{attribute 'qualified_only'}
VAR_GLOBAL  (* GVL_IO *)
  DI_Security_Open : ARRAY[1..GVL_CONSTANTS.C_MAX_SECURITY_SENSORS] OF BOOL;
  DI_Security_Glass : ARRAY[1..GVL_CONSTANTS.C_MAX_SECURITY_SENSORS] OF BOOL;
  DI_Security_2F_Group : BOOL;
  DI_Flood_Sensors : ARRAY[1..GVL_CONSTANTS.C_MAX_FLOOD_SENSORS] OF BOOL;
  DI_Manifold_End_Switches : ARRAY[1..GVL_CONSTANTS.C_MAX_MANIFOLDS] OF BOOL;
  AO_Manifold_Valves : ARRAY[1..GVL_CONSTANTS.C_MAX_MANIFOLDS] OF UINT;
  DO_Manifold_Pumps : ARRAY[1..GVL_CONSTANTS.C_MAX_MANIFOLDS] OF BOOL;
  AI_Manifold_Currents : ARRAY[1..GVL_CONSTANTS.C_MAX_MANIFOLDS] OF INT;
  AI_Manifold_Pressures : ARRAY[1..GVL_CONSTANTS.C_MAX_MANIFOLDS] OF INT;
  AI_Manifold_Temps_Supply : ARRAY[1..GVL_CONSTANTS.C_MAX_MANIFOLDS] OF ST_Owen_Analog_Value;
  AI_Manifold_Temps_Return : ARRAY[1..GVL_CONSTANTS.C_MAX_MANIFOLDS] OF INT;
  AO_Supply_Fans : ARRAY[1..GVL_CONSTANTS.C_MAX_SUPPLY_FANS] OF UINT;
  AO_Exhaust_Fans : ARRAY[1..GVL_CONSTANTS.C_MAX_EXHAUST_FANS] OF UINT;
  AO_Lighting_Levels : ARRAY[1..GVL_CONSTANTS.C_MAX_LIGHT_ZONES] OF UINT;
  AO_Blinds_Positions : ARRAY[1..GVL_CONSTANTS.C_MAX_BLINDS] OF UINT;
  AI_Supply_Temps : ARRAY[1..GVL_CONSTANTS.C_MAX_SUPPLY_TEMPS] OF ST_Owen_Analog_Value;
  AI_Boiler_Modulation : ARRAY[1..GVL_CONSTANTS.C_MAX_BOILERS] OF INT;
  AI_Boiler_Flame_Status : ARRAY[1..GVL_CONSTANTS.C_MAX_BOILERS] OF BOOL;
  DI_Boiler_Error : ARRAY[1..GVL_CONSTANTS.C_MAX_BOILERS] OF BOOL;
  AI_Methane_LEL : ARRAY[1..GVL_CONSTANTS.C_MAX_METHANE_SENSORS] OF ST_Owen_Analog_Value;
  AI_CO_PPM : ARRAY[1..GVL_CONSTANTS.C_MAX_CO_SENSORS] OF REAL;
  DI_Smoke_Sensors : ARRAY[1..GVL_CONSTANTS.C_MAX_SMOKE_SENSORS] OF BOOL;
  AI_Temp_Outdoor : ST_Owen_Analog_Value;
  AI_Floor_Temps : ARRAY[1..GVL_CONSTANTS.C_MAX_ZONES] OF REAL;
  AI_Room_Temps : ARRAY[1..GVL_CONSTANTS.C_MAX_ZONES] OF REAL;
  AI_Room_Hum : ARRAY[1..GVL_CONSTANTS.C_MAX_ZONES] OF REAL;
  AI_Room_CO2 : ARRAY[1..GVL_CONSTANTS.C_MAX_ZONES] OF REAL;
  DO_Zone_Valves : ARRAY[1..GVL_CONSTANTS.C_MAX_HEATING_CIRCUITS] OF BOOL;
  AI_DHW_Temp : REAL;
  AI_DHW_Pressure : REAL;
  DO_DHW_Heating_Pump : BOOL;
  DO_DHW_Circ_Pump : BOOL;
  DO_Backup_Circulation_Pump : BOOL;
  DO_Electric_Heater_Enable : BOOL;
  DI_Lighting_Switches : ARRAY[1..GVL_CONSTANTS.C_MAX_LIGHT_ZONES] OF BOOL;
  DI_Socket_Switches : ARRAY[1..GVL_CONSTANTS.C_MAX_SOCKETS] OF BOOL;
  DI_Motion_Sensors : ARRAY[1..GVL_CONSTANTS.C_MAX_LIGHT_ZONES] OF BOOL;
  DO_Sockets : ARRAY[1..GVL_CONSTANTS.C_MAX_SOCKETS] OF BOOL;
  DO_Gas_Valve_Close : BOOL;
  DO_Water_Valve_35_Close : BOOL;
  DO_Water_Valve_36_Close : BOOL;
  AI_Water_Valve_35_Current : REAL;
  AI_Water_Valve_36_Current : REAL;
  DI_Power_OK : BOOL;
  DO_Gas_Siren : BOOL;
  DO_Fire_Siren : BOOL;
  DO_Security_Siren : BOOL;
  DO_Pump_Main_Enable : BOOL;
  DO_Gate_Open : BOOL;
  DO_Wicket_Open : BOOL;
  DO_Lock_1_Open : BOOL;
  DO_Lock_1_Close : BOOL;
  DO_Lock_2_Open : BOOL;
  DO_Lock_2_Close : BOOL;
  DI_Partner_Pulse : BOOL;
  DI_Partner_Active : BOOL;
  DO_Heartbeat_Pulse : BOOL;
  DO_Active_Status : BOOL;
  DI_Module_1_Heartbeat : BOOL;
  DI_Module_2_Heartbeat : BOOL;
  DI_Backup_Circulation_Pump_Feedback : BOOL;
  DI_Electric_Heater_Feedback : BOOL;
  DI_Water_Zone_Open_FB : ARRAY[1..GVL_CONSTANTS.C_MAX_WATER_ZONES] OF BOOL;
  DI_Water_Zone_Close_FB : ARRAY[1..GVL_CONSTANTS.C_MAX_WATER_ZONES] OF BOOL;
  DO_Water_Zone_Enable : ARRAY[1..GVL_CONSTANTS.C_MAX_WATER_ZONES] OF BOOL;
END_VAR

VAR_GLOBAL  (* GVL_Safety_Selector *)
  G_Use_Shadow_CO : BOOL := FALSE;
  G_Use_Shadow_Methane : BOOL := FALSE;
  G_Use_Shadow_Smoke : BOOL := FALSE;
  G_CO_Effective : REAL;
  G_Methane_Effective : REAL;
  G_Smoke_Effective : BOOL;
  G_CO_Shadow_Max_Diff : REAL := 5.0;
  G_Methane_Shadow_Max_Diff : REAL := 5.0;
  G_Block_Shadow_On_Mismatch : BOOL := TRUE;
  G_Shadow_Unstable_Cycles_Limit : INT := 5;
  G_CO_Shadow_Recovery_Diff : REAL := 2.0;
  G_Methane_Shadow_Recovery_Diff : REAL := 2.0;
  G_CO_Stable_Counter : INT := 0;
  G_Methane_Stable_Counter : INT := 0;
  G_Smoke_Stable_Counter : INT := 0;
  G_CO_Unstable_Counter : INT := 0;
  G_Methane_Unstable_Counter : INT := 0;
  G_Smoke_Unstable_Counter : INT := 0;
  G_CO_Effective_Array : ARRAY[1..GVL_CONSTANTS.C_MAX_CO_SENSORS] OF REAL;
  G_Methane_Effective_Array : ARRAY[1..GVL_CONSTANTS.C_MAX_METHANE_SENSORS] OF REAL;
  G_Smoke_Effective_Array : ARRAY[1..GVL_CONSTANTS.C_MAX_SMOKE_SENSORS] OF BOOL;
END_VAR

{attribute 'qualified_only'}
VAR_GLOBAL  (* GVL_STATE *)
  G_Floor_Temps : ARRAY[1..GVL_CONSTANTS.C_MAX_HEATING_CIRCUITS] OF REAL;
  G_Room_Temps : ARRAY[1..GVL_CONSTANTS.C_MAX_ZONES] OF REAL;
  G_Last_Valid_Room_Temps : ARRAY[1..GVL_CONSTANTS.C_MAX_ZONES] OF REAL;
  G_Last_Valid_Floor_Temps : ARRAY[1..GVL_CONSTANTS.C_MAX_HEATING_CIRCUITS] OF REAL;
  G_Temp_Sensor_Fault : ARRAY[1..GVL_CONSTANTS.C_MAX_ZONES] OF BOOL;
  G_Floor_Temp_Sensor_Fault : ARRAY[1..GVL_CONSTANTS.C_MAX_HEATING_CIRCUITS] OF BOOL;
  G_Room_Hum : ARRAY[1..GVL_CONSTANTS.C_MAX_ZONES] OF REAL;
  G_Room_CO2 : ARRAY[1..GVL_CONSTANTS.C_MAX_ZONES] OF REAL;
  G_Motion_Sensors : ARRAY[1..GVL_CONSTANTS.C_MAX_LIGHT_ZONES] OF BOOL;
  G_Door_Sensors : ARRAY[1..GVL_CONSTANTS.C_MAX_DOOR_SENSORS] OF BOOL;
  G_Window_Sensors : ARRAY[1..GVL_CONSTANTS.C_MAX_ZONES] OF BOOL;
  G_Water_Sensors : ARRAY[1..GVL_CONSTANTS.C_MAX_FLOOD_SENSORS] OF BOOL;
  G_Flood_Warning : ARRAY[1..GVL_CONSTANTS.C_MAX_FLOOD_SENSORS] OF BOOL;
  G_Flood_Alarm : ARRAY[1..GVL_CONSTANTS.C_MAX_FLOOD_SENSORS] OF BOOL;
  G_Flood_Warning_Rise : ARRAY[1..GVL_CONSTANTS.C_MAX_FLOOD_SENSORS] OF BOOL;
  G_Flood_Alarm_Rise : ARRAY[1..GVL_CONSTANTS.C_MAX_FLOOD_SENSORS] OF BOOL;
  G_Flood_Alarm_Fall : ARRAY[1..GVL_CONSTANTS.C_MAX_FLOOD_SENSORS] OF BOOL;
  G_Smoke_Sensors : ARRAY[1..GVL_CONSTANTS.C_MAX_SMOKE_SENSORS] OF BOOL;
  G_Methane_Sensors : ARRAY[1..GVL_CONSTANTS.C_MAX_METHANE_SENSORS] OF REAL;
  G_CO_Sensors : ARRAY[1..GVL_CONSTANTS.C_MAX_CO_SENSORS] OF REAL;
  G_Manifold_Pressures : ARRAY[1..GVL_CONSTANTS.C_MAX_MANIFOLDS] OF REAL;
  G_Manifold_Currents : ARRAY[1..GVL_CONSTANTS.C_MAX_MANIFOLDS] OF REAL;
  G_Predictive_Pump_Pressure_Drop : ARRAY[1..GVL_CONSTANTS.C_MAX_MANIFOLDS] OF BOOL;
  G_Predictive_Pump_Current_Rise : ARRAY[1..GVL_CONSTANTS.C_MAX_MANIFOLDS] OF BOOL;
  G_Manifold_T_Supply : ARRAY[1..GVL_CONSTANTS.C_MAX_MANIFOLDS] OF REAL;
  G_Manifold_T_Return : ARRAY[1..GVL_CONSTANTS.C_MAX_MANIFOLDS] OF REAL;
  G_Boiler_Flame : ARRAY[1..GVL_CONSTANTS.C_MAX_BOILERS] OF BOOL;
  G_Boiler_Error : ARRAY[1..GVL_CONSTANTS.C_MAX_BOILERS] OF BOOL;
  G_Boiler_OT_Online : ARRAY[1..GVL_CONSTANTS.C_MAX_BOILERS] OF BOOL;
  G_Boiler_OT_Command_Ack : ARRAY[1..GVL_CONSTANTS.C_MAX_BOILERS] OF BOOL;
  G_Boiler_OT_Command_Timeout : ARRAY[1..GVL_CONSTANTS.C_MAX_BOILERS] OF BOOL;
  G_Boiler_OT_Heartbeat_Timeout : ARRAY[1..GVL_CONSTANTS.C_MAX_BOILERS] OF BOOL;
  G_Boiler_OT_Adapter_Error : ARRAY[1..GVL_CONSTANTS.C_MAX_BOILERS] OF BOOL;
  G_Boiler_OT_Heartbeat_Age_MS : ARRAY[1..GVL_CONSTANTS.C_MAX_BOILERS] OF UDINT;
  G_Boiler_OT_Command_Age_MS : ARRAY[1..GVL_CONSTANTS.C_MAX_BOILERS] OF UDINT;
  G_Boiler_OT_Adapter_State : ARRAY[1..GVL_CONSTANTS.C_MAX_BOILERS] OF E_OpenTherm_Adapter_State;
  G_Boiler_OT_Error_State : ARRAY[1..GVL_CONSTANTS.C_MAX_BOILERS] OF E_OpenTherm_Error;
  G_Boiler_OT_Enable : ARRAY[1..GVL_CONSTANTS.C_MAX_BOILERS] OF BOOL;
  G_Boiler_OT_Setpoint : ARRAY[1..GVL_CONSTANTS.C_MAX_BOILERS] OF REAL;
  G_Heating_Cascade_Available : BOOL;
  G_Heating_Cascade_Degraded : BOOL;
  G_Heating_Cascade_Partial_Capacity : BOOL;
  G_Heating_Cascade_No_Flame : BOOL;
  G_Heating_Cascade_Transport_Degraded : BOOL;
  G_Heating_Cascade_Ignition_Timeout : BOOL;
  G_Heating_Cascade_Active_Boilers : UINT;
  G_Heating_Cascade_Available_Boilers : UINT;
  G_Physical_Switches : ARRAY[1..GVL_CONSTANTS.C_MAX_LIGHT_ZONES] OF BOOL;
  G_Socket_Switches : ARRAY[1..GVL_CONSTANTS.C_MAX_SOCKETS] OF BOOL;
  G_Outdoor_Temp : REAL;
  G_Supply_Temps : ARRAY[1..GVL_CONSTANTS.C_MAX_SUPPLY_TEMPS] OF REAL;
  G_DHW_Temp : REAL;
  G_DHW_Pressure : REAL;
  G_Zone_Valves : ARRAY[1..GVL_CONSTANTS.C_MAX_HEATING_CIRCUITS] OF BOOL;
  G_Manifold_Pumps : ARRAY[1..GVL_CONSTANTS.C_MAX_MANIFOLDS] OF BOOL;
  G_Manifold_Valves : ARRAY[1..GVL_CONSTANTS.C_MAX_MANIFOLDS] OF REAL;
  G_Manifold_End_Switches : ARRAY[1..GVL_CONSTANTS.C_MAX_MANIFOLDS] OF BOOL;
  G_Supply_Fans : ARRAY[1..GVL_CONSTANTS.C_MAX_SUPPLY_FANS] OF REAL;
  G_Exhaust_Fans : ARRAY[1..GVL_CONSTANTS.C_MAX_EXHAUST_FANS] OF REAL;
  G_Vent_Heater_Power : ARRAY[1..GVL_CONSTANTS.C_MAX_BOILERS] OF REAL;
  G_Lighting_Levels : ARRAY[1..GVL_CONSTANTS.C_MAX_LIGHT_ZONES] OF BYTE;
  G_Blinds_Positions : ARRAY[1..GVL_CONSTANTS.C_MAX_BLINDS] OF BYTE;
  G_Socket_States : ARRAY[1..GVL_CONSTANTS.C_MAX_SOCKETS] OF BOOL;
  G_DHW_Heating_Pump : BOOL;
  G_DHW_Circ_Pump : BOOL;
  G_Backup_Circulation_Pump : BOOL;
  G_Electric_Heater_Enable : BOOL;
  G_Safety_Gas_Alarm : BOOL;
  G_Safety_Leak_Alarm : BOOL;
  G_Safety_Smoke_Alarm : BOOL;
  G_Safety_Emergency_Stop : BOOL;
  G_Safety_Gas_Latched : BOOL;
  G_Safety_Leak_Latched : BOOL;
  G_Safety_Smoke_Latched : BOOL;
  G_Safety_Freeze_Risk : BOOL;
  G_System_Mode : E_System_Operating_Mode := E_System_Operating_Mode.MODE_NORMAL;
  G_System_Mode_Text : STRING(64);
  G_Heating_IO_Fault : BOOL;
  G_Heating_Sensor_Fault : BOOL;
  G_Heating_Subsystem_Degraded : BOOL;
  G_Allocation_Policy_Active : BOOL;
  G_Allocation_Freeze_Bypass_Active : BOOL;
  G_Allocation_DHW_Bypass_Active : BOOL;
  G_Allocation_Budget_Max : REAL;
  G_Allocation_Budget_Used : REAL;
  G_Allocation_Requested : ARRAY[1..GVL_CONSTANTS.C_MAX_MANIFOLDS] OF BOOL;
  G_Allocation_Allowed : ARRAY[1..GVL_CONSTANTS.C_MAX_MANIFOLDS] OF BOOL;
  G_Allocation_Filtered : ARRAY[1..GVL_CONSTANTS.C_MAX_MANIFOLDS] OF BOOL;
  G_Allocation_Block_Reason : ARRAY[1..GVL_CONSTANTS.C_MAX_MANIFOLDS] OF E_Heating_Allocation_Block_Reason;
  G_Allocation_Effective_Priority : ARRAY[1..GVL_CONSTANTS.C_MAX_MANIFOLDS] OF INT;
  G_Policy_Target_Adjustment_Active : BOOL;
  G_Policy_Target_Adjustment_Applied : REAL;
  G_Policy_Priority_Multiplier_Applied : REAL;
  G_Policy_Priority_Bridge_Active : BOOL;
  G_Policy_Priority_Bias_Applied : ARRAY[1..GVL_CONSTANTS.C_MAX_MANIFOLDS] OF REAL;
  G_Policy_Priority_Effective : ARRAY[1..GVL_CONSTANTS.C_MAX_MANIFOLDS] OF INT;
  G_Heating_RootCause : E_Heating_RootCause := E_Heating_RootCause.RC_NONE;
  G_Heating_RootConfidence : REAL;
  G_Heating_Confidence : REAL := 1.0;
  G_Heating_Error_Score : REAL := 0.0;
  G_Heating_Confidence_Reason_Code : INT := 0;
  G_Heating_Confidence_Reason_Text : STRING(128) := 'OK';
  G_DHW_IO_Fault : BOOL;
  G_DHW_Sensor_Fault : BOOL;
  G_DHW_Subsystem_Degraded : BOOL;
  G_Ventilation_IO_Fault : BOOL;
  G_Ventilation_Subsystem_Degraded : BOOL;
  G_Lighting_IO_Fault : BOOL;
  G_Lighting_Subsystem_Degraded : BOOL;
  G_Access_Comm_Fault : BOOL;
  G_Evacuation_Lighting_Active : BOOL;
  G_Evac_Hazard_Zone : ARRAY[1..GVL_CONSTANTS.C_MAX_LIGHT_ZONES] OF BOOL;
  G_Evac_Guidance : ARRAY[1..GVL_CONSTANTS.C_MAX_LIGHT_ZONES] OF INT;
  G_Rule_Actions : ARRAY[1..GVL_CONSTANTS.C_MAX_RULES] OF ST_Rule_Action;
  G_Sim_Lights : ARRAY[1..GVL_CONSTANTS.C_MAX_LIGHT_ZONES] OF BOOL;
  G_Freeze_Hardware_Degraded : BOOL;
  G_Freeze_Hardware_Failed : BOOL;
  G_Water_Zone_Enable : ARRAY[1..GVL_CONSTANTS.C_MAX_WATER_ZONES] OF BOOL;
  G_Water_Zone_Open_FB : ARRAY[1..GVL_CONSTANTS.C_MAX_WATER_ZONES] OF BOOL;
  G_Water_Zone_Close_FB : ARRAY[1..GVL_CONSTANTS.C_MAX_WATER_ZONES] OF BOOL;
  G_Water_Zone_Exercise_Active : ARRAY[1..GVL_CONSTANTS.C_MAX_WATER_ZONES] OF BOOL;
  G_Preheat_Request : BOOL;
  G_Freeze_Request : BOOL;
  G_Target_Temperature : REAL;
END_VAR

VAR_GLOBAL  (* GVL_TRANSPORT_FRESHNESS *)
  Transport_Epoch : ULINT := 0;
  Transport_Publication_Epoch : ULINT := 0;
  Transport_Freshness_Valid : BOOL := FALSE;
  Transport_Publication_Allowed : BOOL := FALSE;
  Transport_Lease_Valid : BOOL := FALSE;
  Transport_Lease_Expired : BOOL := FALSE;
  Transport_Lease_Timeout_MS : UDINT := 5000;
  Transport_Quarantine_Active : BOOL := FALSE;
  Transport_Reconnect_Stabilizing : BOOL := FALSE;
  Transport_Stale_Frame_Detected : BOOL := FALSE;
  Transport_Transaction_Mismatch : BOOL := FALSE;
  Transport_Snapshot_Invalid : BOOL := FALSE;
  Transport_Last_Refresh_MS : UDINT := 0;
  Transport_Last_Reconnect_MS : UDINT := 0;
  Transport_Last_Publication_MS : UDINT := 0;
  Transport_Last_Error_Code : UDINT := 0;
  Transport_Last_Error_Text : STRING(160) := '';
  Transport_Invalidation_Count : UDINT := 0;
END_VAR

{attribute 'qualified_only'}
VAR_GLOBAL  (* GVL_Heating_Circuit_Explainability *)
  G_Source_Selection_Visible : ARRAY[1..GVL_CONSTANTS.C_MAX_HEATING_CIRCUITS] OF BOOL;
  G_Selected_Source_Code : ARRAY[1..GVL_CONSTANTS.C_MAX_HEATING_CIRCUITS] OF UINT;  (* 0 none, 1 room, 2 floor *)
  G_Selected_Source_Text : ARRAY[1..GVL_CONSTANTS.C_MAX_HEATING_CIRCUITS] OF STRING(64);
  G_Fallback_Active : ARRAY[1..GVL_CONSTANTS.C_MAX_HEATING_CIRCUITS] OF BOOL;
  G_Source_Degraded : ARRAY[1..GVL_CONSTANTS.C_MAX_HEATING_CIRCUITS] OF BOOL;
  G_Selected_Source_Confidence : ARRAY[1..GVL_CONSTANTS.C_MAX_HEATING_CIRCUITS] OF REAL;
  G_Primary_Source_Confidence : ARRAY[1..GVL_CONSTANTS.C_MAX_HEATING_CIRCUITS] OF REAL;
  G_Fallback_Source_Confidence : ARRAY[1..GVL_CONSTANTS.C_MAX_HEATING_CIRCUITS] OF REAL;
  G_Reason_Code : ARRAY[1..GVL_CONSTANTS.C_MAX_HEATING_CIRCUITS] OF UINT;  (* 0 OK, 1 primary degraded fallback used, 2 degraded primary retained, 3 source loss *)
  G_Reason_Text : ARRAY[1..GVL_CONSTANTS.C_MAX_HEATING_CIRCUITS] OF STRING(128);
  G_Source_Switched_Event : ARRAY[1..GVL_CONSTANTS.C_MAX_HEATING_CIRCUITS] OF BOOL;
  G_Fallback_Activated_Event : ARRAY[1..GVL_CONSTANTS.C_MAX_HEATING_CIRCUITS] OF BOOL;
  G_Fallback_Recovered_Event : ARRAY[1..GVL_CONSTANTS.C_MAX_HEATING_CIRCUITS] OF BOOL;
  G_Source_Loss_Event : ARRAY[1..GVL_CONSTANTS.C_MAX_HEATING_CIRCUITS] OF BOOL;
  G_Last_Event_MS : ARRAY[1..GVL_CONSTANTS.C_MAX_HEATING_CIRCUITS] OF UDINT;
  G_Last_Event_Code : ARRAY[1..GVL_CONSTANTS.C_MAX_HEATING_CIRCUITS] OF UINT;  (* 0 none, 1 switched, 2 fallback activated, 3 fallback recovered, 4 source loss *)
  G_Last_Event_Text : ARRAY[1..GVL_CONSTANTS.C_MAX_HEATING_CIRCUITS] OF STRING(128);
END_VAR

{attribute 'qualified_only'}
VAR_GLOBAL  (* GVL_Water_Hydraulic_Topology *)
  G_Topology_Node : ARRAY[1..64] OF ST_Water_Hydraulic_Topology_Node;
  G_Isolation_Group : ARRAY[1..64] OF ST_Water_Hydraulic_Isolation_Group;
  G_Any_Ambiguous : BOOL;
  G_Any_Global_Fallback_Required : BOOL;
  G_Runtime_Valid : BOOL;
  G_Last_Update_MS : UDINT;
  G_Status_Code : UINT;
  G_Status_Text : STRING(128);
END_VAR

VAR_GLOBAL  (* GVL_RECOVERY_GOVERNANCE *)
  Recovery_Epoch : ULINT := 0;
  Recovery_Cleanup_Epoch : ULINT := 0;
  Recovery_Governance_Valid : BOOL := FALSE;
  Recovery_Cleanup_Completed : BOOL := FALSE;
  Recovery_Cleanup_Verified : BOOL := FALSE;
  Recovery_Quarantine_Active : BOOL := FALSE;
  Recovery_Forced_Safe_Mode : BOOL := FALSE;
  Recovery_Semantic_Residue_Detected : BOOL := FALSE;
  Recovery_Degraded_State_Residual : BOOL := FALSE;
  Recovery_Retained_State_Residual : BOOL := FALSE;
  Recovery_Last_Cleanup_Start_MS : UDINT := 0;
  Recovery_Last_Cleanup_End_MS : UDINT := 0;
  Recovery_Last_Error_Code : UDINT := 0;
  Recovery_Last_Error_Text : STRING(160) := '';
  Recovery_Invalidation_Count : UDINT := 0;
END_VAR

VAR_GLOBAL  (* GVL_SEMANTIC_PRESERVATION_FABRIC *)
  Semantic_Preservation_Valid : BOOL := FALSE;
  Semantic_Preservation_Granted : BOOL := FALSE;
  Semantic_Preservation_Quarantine_Active : BOOL := TRUE;
  Declared_System_Intent_Coherent : BOOL := FALSE;
  Adaptive_Policy_Bounded : BOOL := FALSE;
  Cross_Domain_Intent_Aligned : BOOL := FALSE;
  Optimization_Goals_Coherent : BOOL := FALSE;
  Behavioral_Evolution_Stable : BOOL := FALSE;
  Objective_Boundaries_Immutable : BOOL := FALSE;
  Semantic_Governance_Coherent : BOOL := FALSE;
  Adaptive_Runtime_Intent_Stable : BOOL := FALSE;
  LongTerm_Semantic_Evolution_Valid : BOOL := FALSE;
  Adaptive_Policy_Drift_Detected : BOOL := FALSE;
  Optimization_Semantic_Erosion_Detected : BOOL := FALSE;
  CrossDomain_Intent_Divergence_Detected : BOOL := FALSE;
  LongTerm_Objective_Mutation_Detected : BOOL := FALSE;
  Behavior_Learning_Instability_Detected : BOOL := FALSE;
  Silent_Governance_Reinterpretation_Detected : BOOL := FALSE;
  Semantic_Preservation_Epoch : UDINT := 0;
  Semantic_Preservation_Epoch_Coherent : BOOL := FALSE;
  Semantic_Preservation_Last_Update_MS : UDINT := 0;
  Semantic_Preservation_Lease_Expired : BOOL := TRUE;
  Semantic_Preservation_Last_Error_Code : UDINT := 0;
  Semantic_Preservation_Last_Error_Text : STRING(160) := '';
  Semantic_Preservation_Invalidation_Count : UDINT := 0;
END_VAR

VAR_GLOBAL  (* GVL_OBSERVABILITY_AUTHORITY *)
  Observability_Epoch : ULINT := 0;
  Observability_Snapshot_Epoch : ULINT := 0;
  Publication_Runtime_Valid : BOOL := FALSE;
  Unsafe_State_Published : BOOL := FALSE;
  Emergency_Visibility_Required : BOOL := FALSE;
  Runtime_Failure_Visible : BOOL := FALSE;
  Output_Decay_Visible : BOOL := FALSE;
  Transport_Failure_Visible : BOOL := FALSE;
  Recovery_Failure_Visible : BOOL := FALSE;
  Fencing_Failure_Visible : BOOL := FALSE;
  Monotonic_Failure_Visible : BOOL := FALSE;
  Distributed_Failure_Visible : BOOL := FALSE;
  Distributed_Quarantine_Visible : BOOL := FALSE;
  Peer_Runtime_Stale_Visible : BOOL := FALSE;
  Peer_Snapshot_Stale_Visible : BOOL := FALSE;
  Peer_Boot_Mismatch_Visible : BOOL := FALSE;
  Peer_Fencing_Conflict_Visible : BOOL := FALSE;
  Peer_Semantic_Continuity_Lost_Visible : BOOL := FALSE;
  Distributed_Publication_Reconciliation_Visible : BOOL := FALSE;
  Distributed_Publication_Freeze_Visible : BOOL := FALSE;
  Distributed_Snapshot_Consistency_Visible : BOOL := FALSE;
  Peer_Publication_Stale_Visible : BOOL := FALSE;
  Peer_Publication_Divergence_Visible : BOOL := FALSE;
  Peer_Publication_Reconciliation_Lost_Visible : BOOL := FALSE;
  Peer_Snapshot_Not_Immutable_Visible : BOOL := FALSE;
  Distributed_Immutable_Snapshot_Quarantine_Visible : BOOL := FALSE;
  Distributed_Commit_Visible : BOOL := FALSE;
  Distributed_Commit_Quarantine_Visible : BOOL := FALSE;
  Publication_Prepare_Visible : BOOL := FALSE;
  Publication_Commit_Visible : BOOL := FALSE;
  Peer_Commit_Ack_Visible : BOOL := FALSE;
  Peer_Commit_Mismatch_Visible : BOOL := FALSE;
  Peer_Commit_Replay_Visible : BOOL := FALSE;
  Peer_Commit_Missing_Visible : BOOL := FALSE;
  Commit_Lease_Expired_Visible : BOOL := FALSE;
  Observability_Last_Publication_MS : UDINT := 0;
  Observability_Last_Error_Code : UDINT := 0;
  Observability_Last_Error_Text : STRING(160) := '';
END_VAR

VAR_GLOBAL  (* GVL_CAUSALITY_REVERSAL_PREVENTION_FABRIC *)
  Causality_Reversal_Prevention_Valid : BOOL := FALSE;
  Causality_Reversal_Prevention_Granted : BOOL := FALSE;
  Causality_Reversal_Prevented : BOOL := FALSE;
  Authority_Ordering_Canonical : BOOL := FALSE;
  Revocation_Resurrection_Boundary_Stable : BOOL := FALSE;
  Reversal_Causality_Grounded : BOOL := FALSE;
  Distributed_Reversal_Consensus_Valid : BOOL := FALSE;
  Causality_Reversal_Detected : BOOL := FALSE;
  Resurrection_After_Revocation_Detected : BOOL := FALSE;
  Unsafe_Temporal_Replay_Detected : BOOL := FALSE;
  Causality_Reversal_Epoch : UDINT := 0;
END_VAR

VAR_GLOBAL  (* GVL_ACTUATOR_SEMANTIC_VERIFICATION *)
  Actuator_Semantic_Verification_Valid : BOOL := FALSE;
  Actuator_Semantic_Verification_Granted : BOOL := FALSE;
  Actuator_Semantic_Verification_Quarantine_Active : BOOL := TRUE;
  Valve_Semantic_Realization_Valid : BOOL := FALSE;
  Relay_Semantic_Realization_Valid : BOOL := FALSE;
  Pump_Semantic_Realization_Valid : BOOL := FALSE;
  Fan_Semantic_Realization_Valid : BOOL := FALSE;
  Hydraulic_Response_Valid : BOOL := FALSE;
  Physical_Effect_Converged : BOOL := FALSE;
  Actuation_Response_Temporal_Valid : BOOL := FALSE;
  Sensor_Confirmed_Execution_Valid : BOOL := FALSE;
  Semantic_Outcome_Aligned : BOOL := FALSE;
  False_Positive_Actuation_Detected : BOOL := FALSE;
  Mechanical_NonRealization_Detected : BOOL := FALSE;
  Welded_Relay_Semantics_Detected : BOOL := FALSE;
  Hydraulic_NoEffect_Execution_Detected : BOOL := FALSE;
  Airflow_Realization_Mismatch_Detected : BOOL := FALSE;
  Physical_Convergence_Divergence_Detected : BOOL := FALSE;
  Actuator_Verification_Epoch : UDINT := 0;
  Actuator_Verification_Epoch_Coherent : BOOL := FALSE;
  Actuator_Verification_Last_Update_MS : UDINT := 0;
  Actuator_Verification_Lease_Expired : BOOL := TRUE;
  Actuator_Verification_Last_Error_Code : UDINT := 0;
  Actuator_Verification_Last_Error_Text : STRING(160) := '';
  Actuator_Verification_Invalidation_Count : UDINT := 0;
END_VAR

VAR_GLOBAL  (* GVL_INPUT_QUALITY *)
  G_Room_Temp_Quality : ARRAY[1..16] OF ST_Input_Quality_Record;
  G_Floor_Temp_Quality : ARRAY[1..GVL_CONSTANTS.C_MAX_HEATING_CIRCUITS] OF ST_Input_Quality_Record;
END_VAR

VAR_GLOBAL  (* GVL_RUNTIME_BUDGET_ENFORCEMENT *)
  Runtime_Budget_Enforcement_Active : BOOL := TRUE;
  Runtime_Budget_Enforcement_ReadOnly : BOOL := TRUE;
  Verification_Runtime_Budget_Observed : BOOL := FALSE;
  Observability_Runtime_Budget_Observed : BOOL := FALSE;
  Diagnostics_Runtime_Budget_Observed : BOOL := FALSE;
  Governance_Runtime_Overhead_Observed : BOOL := FALSE;
  Runtime_Budget_Pressure_Observed : BOOL := FALSE;
  Verification_Time_Budget_Exceeded : BOOL := FALSE;
  Observability_Amplification_Budget_Exceeded : BOOL := FALSE;
  Diagnostics_Load_Budget_Exceeded : BOOL := FALSE;
  Runtime_Stability_Budget_At_Risk : BOOL := FALSE;
  Verification_Induced_Runtime_Risk : BOOL := FALSE;
  Runtime_Budget_Enforcement_Epoch : UDINT := 0;
END_VAR

{attribute 'qualified_only'}
VAR_GLOBAL  (* GVL_GATEWAY *)
  G_Gateway_Command : ST_Gateway_Command;
  G_Gateway_Command_Received : BOOL;
  G_Gateway_Send_2FA : BOOL;
  G_Gateway_2FA_Code : STRING(6);
  G_Gateway_Telegram_Msg : STRING(200);
  G_Gateway_Send_Telegram : BOOL;
  G_Gateway_HMI_Status_Message : STRING(200);
  G_Gateway_Ping_OK : BOOL;
  G_Gateway_Data_Ready : BOOL;
  G_Gateway_Modbus_Registers : ARRAY[0..GVL_CONSTANTS.C_MAX_MODBUS_REGISTERS-1] OF WORD;
  G_Shadow_Alert_Active : BOOL;
  G_Shadow_Dominant_Channel : STRING(32);
  G_Shadow_Policy_Summary_Text : STRING(160);
  G_Shadow_Recent_Activity_Text : STRING(160);
  G_Shadow_Rate_Summary_Text : STRING(160);
  G_Shadow_Total_Fallback_Count : UDINT;
  G_Shadow_Total_Recovery_Count : UDINT;
END_VAR

{attribute 'qualified_only'}
VAR_GLOBAL  (* GVL_Water_Physical_Runtime *)
  G_Convergence_State : ARRAY[1..64] OF ST_Water_Physical_Convergence_State;
  G_Actuator_Diagnostics : ARRAY[1..64] OF ST_Water_Actuator_Diagnostics_State;
  G_Any_Convergence_Degraded : BOOL;
  G_Any_Diagnostics_Degraded : BOOL;
  G_Any_Escalation_Required : BOOL;
  G_Runtime_Valid : BOOL;
  G_Last_Update_MS : UDINT;
  G_Status_Code : UINT;
  G_Status_Text : STRING(128);
END_VAR

{attribute 'qualified_only'}
VAR_GLOBAL  (* GVL_Runtime_Discovery *)
  G_Discovery_State : ARRAY[1..32] OF ST_Runtime_Node_Discovery_State;
END_VAR

VAR_GLOBAL  (* GVL_FORENSIC_EVIDENCE_FABRIC *)
  Forensic_Evidence_Valid : BOOL := FALSE;
  Forensic_Evidence_Granted : BOOL := FALSE;
  Forensic_Evidence_Quarantine_Active : BOOL := TRUE;
  Authority_Lineage_Reconstructable : BOOL := FALSE;
  Decision_Causality_Traceable : BOOL := FALSE;
  Distributed_Evidence_Coherent : BOOL := FALSE;
  Immutable_Audit_Continuity_Valid : BOOL := FALSE;
  Recovery_Lineage_Preserved : BOOL := FALSE;
  Historical_Proof_Chain_Valid : BOOL := FALSE;
  Governance_Event_Lineage_Coherent : BOOL := FALSE;
  Semantic_Transition_Traceable : BOOL := FALSE;
  Physical_Transition_Traceable : BOOL := FALSE;
  Authority_Lineage_Gap_Detected : BOOL := FALSE;
  NonReconstructable_Decision_Detected : BOOL := FALSE;
  History_Evidence_Divergence_Detected : BOOL := FALSE;
  Causal_Chain_Erosion_Detected : BOOL := FALSE;
  Distributed_Forensic_Inconsistency_Detected : BOOL := FALSE;
  Immutable_Audit_Discontinuity_Detected : BOOL := FALSE;
  Forensic_Evidence_Epoch : UDINT := 0;
  Forensic_Evidence_Epoch_Coherent : BOOL := FALSE;
  Forensic_Evidence_Last_Update_MS : UDINT := 0;
  Forensic_Evidence_Lease_Expired : BOOL := TRUE;
  Forensic_Evidence_Last_Error_Code : UDINT := 0;
  Forensic_Evidence_Last_Error_Text : STRING(160) := '';
  Forensic_Evidence_Invalidation_Count : UDINT := 0;
END_VAR

{attribute 'qualified_only'}
VAR_GLOBAL  (* GVL_SYSTEM_COORDINATION *)
  G_System_Degraded : BOOL := FALSE;
  G_Block_Heating : BOOL := FALSE;
  G_Block_Ventilation : BOOL := FALSE;
  G_Block_Lighting_Override : BOOL := FALSE;
  G_Block_Sockets_Override : BOOL := FALSE;
  G_Coordination_Code : UDINT := 0;
  G_Coordination_Status_Msg : STRING(200) := '';
END_VAR

{attribute 'qualified_only'}
VAR_GLOBAL  (* GVL_Water_Leak_Explainability *)
  G_Leak_Visible : ARRAY[1..GVL_CONSTANTS.C_MAX_FLOOD_SENSORS] OF BOOL;
  G_Warning_Visible : ARRAY[1..GVL_CONSTANTS.C_MAX_FLOOD_SENSORS] OF BOOL;
  G_Mapping_Valid : ARRAY[1..GVL_CONSTANTS.C_MAX_FLOOD_SENSORS] OF BOOL;
  G_Selectively_Isolatable : ARRAY[1..GVL_CONSTANTS.C_MAX_FLOOD_SENSORS] OF BOOL;
  G_Global_Fallback_Required : ARRAY[1..GVL_CONSTANTS.C_MAX_FLOOD_SENSORS] OF BOOL;
  G_Leak_Confidence : ARRAY[1..GVL_CONSTANTS.C_MAX_FLOOD_SENSORS] OF REAL;
  G_Valve_Group_Id : ARRAY[1..GVL_CONSTANTS.C_MAX_FLOOD_SENSORS] OF UINT;
  G_Hydraulic_Zone_Id : ARRAY[1..GVL_CONSTANTS.C_MAX_FLOOD_SENSORS] OF UINT;
  G_Reason_Code : ARRAY[1..GVL_CONSTANTS.C_MAX_FLOOD_SENSORS] OF UINT;
  G_Reason_Text : ARRAY[1..GVL_CONSTANTS.C_MAX_FLOOD_SENSORS] OF STRING(128);
  G_Warning_Started_Event : ARRAY[1..GVL_CONSTANTS.C_MAX_FLOOD_SENSORS] OF BOOL;
  G_Leak_Confirmed_Event : ARRAY[1..GVL_CONSTANTS.C_MAX_FLOOD_SENSORS] OF BOOL;
  G_Leak_Cleared_Event : ARRAY[1..GVL_CONSTANTS.C_MAX_FLOOD_SENSORS] OF BOOL;
  G_Explainability_Valid : BOOL;
  G_Explainability_Status_Code : UINT;
  G_Explainability_Status_Text : STRING(128);
END_VAR

VAR_GLOBAL  (* GVL_PHYSICAL_DEADLOCK_RESOLUTION_FABRIC *)
  Physical_Deadlock_Resolution_Valid : BOOL := FALSE;
  Physical_Deadlock_Resolution_Granted : BOOL := FALSE;
  Deadlock_Resolution_Canonical : BOOL := FALSE;
  Physical_Forward_Progress_Valid : BOOL := FALSE;
  CrossDomain_Execution_Progress_Stable : BOOL := FALSE;
  Recovery_Progress_Stable : BOOL := FALSE;
  Deadlock_Causality_Grounded : BOOL := FALSE;
  Distributed_Deadlock_Consensus_Valid : BOOL := FALSE;
  Physical_CircularWait_Detected : BOOL := FALSE;
  CrossDomain_Progress_Deadlock : BOOL := FALSE;
  Recovery_Livelock_Detected : BOOL := FALSE;
  Physical_Progress_Stall_Detected : BOOL := FALSE;
  Physical_Deadlock_Resolution_Epoch : UDINT := 0;
END_VAR

VAR_GLOBAL  (* GVL_DISTRIBUTED_EPOCH_LINEARITY_FABRIC *)
  Distributed_Epoch_Linearity_Valid : BOOL := FALSE;
  Distributed_Epoch_Linearity_Granted : BOOL := FALSE;
  Distributed_Epoch_Linearity_Valid_Proof : BOOL := FALSE;
  Epoch_Timeline_Monotonic : BOOL := FALSE;
  Cluster_Epoch_Consensus_Stable : BOOL := FALSE;
  Epoch_Causality_Grounded : BOOL := FALSE;
  Distributed_Epoch_Lineage_Coherent : BOOL := FALSE;
  Epoch_Rollback_Detected : BOOL := FALSE;
  Distributed_Epoch_Fork_Detected : BOOL := FALSE;
  Stale_Epoch_Application_Detected : BOOL := FALSE;
  Distributed_Epoch_Linearity_Epoch : UDINT := 0;
END_VAR

VAR_GLOBAL  (* GVL_TRUST_EPOCH_MONOTONICITY_FABRIC *)
  Trust_Epoch_Monotonicity_Valid : BOOL := FALSE;
  Trust_Epoch_Monotonicity_Granted : BOOL := FALSE;
  Trust_Epoch_Monotonicity_Quarantine_Active : BOOL := TRUE;
  Global_Trust_Epoch_Monotonic : BOOL := FALSE;
  Rollback_Resistant_Authority_Valid : BOOL := FALSE;
  Recovery_Epoch_Strictly_Newer : BOOL := FALSE;
  Distributed_Trust_Vector_Coherent : BOOL := FALSE;
  Irreversible_Trust_Progression_Stable : BOOL := FALSE;
  CrossNode_Trust_Epoch_Aligned : BOOL := FALSE;
  Recovery_Timeline_Dominance_Valid : BOOL := FALSE;
  Federation_Epoch_Progression_Coherent : BOOL := FALSE;
  Trust_Revocation_History_Monotonic : BOOL := FALSE;
  Temporal_Trust_Rollback_Detected : BOOL := FALSE;
  Replay_Authority_Epoch_Detected : BOOL := FALSE;
  CrossNode_Trust_Vector_Regression : BOOL := FALSE;
  Stale_Federation_Epoch_Rejoin : BOOL := FALSE;
  Recovery_Timeline_Fork_Detected : BOOL := FALSE;
  Revoked_Epoch_Resurrection_Detected : BOOL := FALSE;
  Trust_Epoch_Monotonicity_Epoch : UDINT := 0;
  Trust_Epoch_Monotonicity_Epoch_Coherent : BOOL := FALSE;
  Trust_Epoch_Monotonicity_Last_Update_MS : UDINT := 0;
  Trust_Epoch_Monotonicity_Lease_Expired : BOOL := TRUE;
  Trust_Epoch_Monotonicity_Last_Error_Code : UDINT := 0;
  Trust_Epoch_Monotonicity_Last_Error_Text : STRING(160) := '';
  Trust_Epoch_Monotonicity_Invalidation_Count : UDINT := 0;
END_VAR

VAR_GLOBAL  (* GVL_RUNTIME_TRANSITION_SYSTEM *)
  Current_Transition_Result : E_RUNTIME_TRANSITION_RESULT := TRANSITION_VALID;
  Runtime_Transition_Validation_Active : BOOL := TRUE;
  Runtime_Transition_ReadOnly_Mode : BOOL := TRUE;
  Runtime_Transition_NoMutation : BOOL := TRUE;
  Runtime_Transition_Legal : BOOL := FALSE;
  Runtime_Transition_Proofs_Valid : BOOL := FALSE;
  Runtime_Transition_Lineage_Valid : BOOL := FALSE;
  Runtime_Transition_Temporal_Valid : BOOL := FALSE;
  Illegal_Runtime_Transition_Observed : BOOL := FALSE;
  Unsafe_State_Promotion_Observed : BOOL := FALSE;
  Recovery_Without_Lineage_Observed : BOOL := FALSE;
  Unsafe_Trust_Escalation_Observed : BOOL := FALSE;
  Runtime_Transition_Epoch : UDINT := 0;
END_VAR

{attribute 'qualified_only'}
VAR_GLOBAL  (* GVL_Runtime_Restart_Continuity *)
  G_Last_Stable_Config_Version : UDINT;
  G_Last_Known_Runtime_Healthy : BOOL;
  G_Last_Known_Quarantine_State : BOOL;
  G_Restore_Request : BOOL;
  G_Post_Restart_Validation_Request : BOOL;
END_VAR

VAR_GLOBAL  (* GVL_TEMPORAL_CAUSALITY_CLOSURE_FABRIC *)
  Temporal_Causality_Closure_Valid : BOOL := FALSE;
  Temporal_Causality_Closure_Granted : BOOL := FALSE;
  Temporal_Causality_Coherent : BOOL := FALSE;
  Monotonic_Reality_Timeline_Valid : BOOL := FALSE;
  Distributed_Temporal_Alignment_Stable : BOOL := FALSE;
  Recovery_Revocation_Ordering_Valid : BOOL := FALSE;
  Temporal_Causality_Lineage_Coherent : BOOL := FALSE;
  Distributed_Temporal_Consensus_Valid : BOOL := FALSE;
  Temporal_Fork_Detected : BOOL := FALSE;
  Stale_Causality_Application_Detected : BOOL := FALSE;
  Recovery_Before_Revocation_Detected : BOOL := FALSE;
  Distributed_Timeline_Drift_Detected : BOOL := FALSE;
  Temporal_Causality_Epoch : UDINT := 0;
END_VAR

VAR_GLOBAL  (* GVL_PHYSICAL_SNAPSHOT *)
  Physical_Snapshot_Valid : BOOL := FALSE;
  Physical_Snapshot_Frozen : BOOL := FALSE;
  Physical_Snapshot_Publication_Allowed : BOOL := FALSE;
  Physical_Snapshot_Isolation_Valid : BOOL := FALSE;
  Physical_Snapshot_Copy_Valid : BOOL := FALSE;
  Physical_Snapshot_Epoch : UDINT := 0;
  Physical_Snapshot_Runtime_Epoch : UDINT := 0;
  Physical_Snapshot_Output_Epoch : UDINT := 0;
  Physical_Snapshot_Mutation_Detected : BOOL := FALSE;
  Physical_Snapshot_Replay_Suspected : BOOL := FALSE;
  Physical_Snapshot_Lease_Expired : BOOL := TRUE;
  Physical_Snapshot_Consensus_Coherent : BOOL := FALSE;
  Physical_Snapshot_Causality_Coherent : BOOL := FALSE;
  Physical_Snapshot_Last_Update_MS : UDINT := 0;
  Physical_Snapshot_Freshness_Valid : BOOL := FALSE;
  Physical_Snapshot_Last_Error_Code : UDINT := 0;
  Physical_Snapshot_Last_Error_Text : STRING(160) := '';
  Physical_Snapshot_Invalidation_Count : UDINT := 0;
END_VAR

{attribute 'qualified_only'}
VAR_GLOBAL  (* GVL_STATUS *)
  G_System_Time_MS : UDINT;
  G_Last_System_Time_MS : UDINT := 0;
  G_Time_Of_Day_MS : UDINT := 0;
  G_Current_Day : UINT := 1;
  G_Day_Of_Year : UINT := 1;
  G_Current_TOD : TOD;
  G_Current_Scenario : E_SCENARIO_TYPE := E_SCENARIO_TYPE.SCENARIO_NONE;
  G_Previous_Scenario : E_SCENARIO_TYPE := E_SCENARIO_TYPE.SCENARIO_NONE;
  G_Is_Night : BOOL;
  G_PLC_ID : BYTE := 1;
  G_Is_Active_PLC : BOOL;
  G_Other_PLC_Is_Active : BOOL;
  G_Remote_PLC_Last_Seen_MS : UDINT;
  G_Remote_PLC_Alive : BOOL;
  G_Local_PLC_ID : BYTE := 1;
  G_Active_PLC_ID : BYTE := 1;
  G_Remote_PLC_Pulse : BOOL;
  G_Security_Status_Msg : STRING(200);
  G_Gas_Status_Msg : STRING(200);
  G_Flood_Status_Msg : STRING(200);
  G_Vent_Status_Msg : STRING(200);
  G_DHW_Status : ST_DHW_Status;
  G_Manifold_Status : ARRAY[1..GVL_CONSTANTS.C_MAX_MANIFOLDS] OF ST_Manifold_Status;
  G_Boiler_Status : ARRAY[1..GVL_CONSTANTS.C_MAX_BOILERS] OF ST_Boiler_Status;
  G_IO_Modules_Online : ARRAY[1..GVL_CONSTANTS.C_MAX_MODULES] OF BOOL;
  G_Sim_Active : BOOL;
  G_Wet_Zone_Light_Active : BOOL;
  G_System_Mode_Msg : STRING(200);
  G_System_Mode_Cause : STRING(200);
  G_System_Mode_Text : STRING(200);
  G_Evac_Target_Zone_Name : STRING(80);
  G_Evac_Hazard_Zone_Name : STRING(80);
  G_Diagnostics : ST_System_Diagnostics;
  G_Diagnostics_Events : ARRAY[1..50] OF ST_Diagnostic_Event;
  G_Diagnostics_Count : INT := 0;
END_VAR

{attribute 'qualified_only'}
VAR_GLOBAL  (* GVL_MODBUS_RTU_FRAME *)
  G_TX_Frame : ST_Modbus_RTU_Frame;
  G_RX_Frame : ST_Modbus_RTU_Frame;
  G_TX_Ready : BOOL := FALSE;
  G_RX_Ready : BOOL := FALSE;
  G_Last_TX_MS : UDINT := 0;
  G_Last_RX_MS : UDINT := 0;
END_VAR

{attribute 'qualified_only'}
VAR_GLOBAL  (* GVL_INPUT_VALIDATION_CONFIG *)
  G_Enable_Input_Validation : BOOL := TRUE;
  G_Enable_Temporal_Anomaly_Detection : BOOL := TRUE;
  G_Enable_Reputation_Learning : BOOL := TRUE;
  G_Room_Temp_Min : REAL := -40.0;
  G_Room_Temp_Max : REAL := 80.0;
  G_Room_Hum_Min : REAL := 0.0;
  G_Room_Hum_Max : REAL := 100.0;
  G_Room_Temp_Spike_Threshold : REAL := 5.0;
  G_Room_Hum_Spike_Threshold : REAL := 20.0;
  G_Room_Temp_Stuck_Epsilon : REAL := 0.01;
  G_Room_Hum_Stuck_Epsilon : REAL := 0.1;
  G_Sensor_Stuck_Timeout_MS : UDINT := 600000;
  G_Condensation_Hum_Threshold : REAL := 90.0;
  G_Condensation_Temp_Threshold : REAL := 0.0;
  G_Reputation_Learning_Rate : REAL := 0.05;
  G_Reputation_Recovery_Decay : REAL := 0.01;
  G_Min_Sensor_Confidence : REAL := 0.1;
  G_Bad_Spike_Confidence : REAL := 0.3;
  G_Bad_Stuck_Confidence : REAL := 0.2;
  G_Default_Confidence : REAL := 1.0;
END_VAR

{attribute 'qualified_only'}
VAR_GLOBAL CONSTANT  (* GVL_CONSTANTS *)
  C_MAX_ZONES : INT := 16;
  C_MAX_LIGHTING_ZONES : INT := 32;
  C_MAX_HEATING_CIRCUITS : INT := 16;
  C_MAX_CLIMATE_ZONES : INT := 16;
  C_MAX_LIGHT_ZONES : INT := 32;
  C_MAX_SOCKETS : INT := 36;
  C_MAX_BLINDS : INT := 20;
  C_MAX_ALARMS : INT := 20;
  C_MAX_RULES : INT := 20;
  C_MAX_MANIFOLDS : INT := 5;
  C_MAX_BOILERS : INT := 2;
  C_MAX_SUPPLY_FANS : INT := 3;
  C_MAX_EXHAUST_FANS : INT := 5;
  C_MAX_SECURITY_SENSORS : INT := 15;
  C_MAX_FLOOD_SENSORS : INT := 12;
  C_MAX_DOOR_SENSORS : INT := 8;
  C_MAX_CO_SENSORS : INT := 8;
  C_MAX_METHANE_SENSORS : INT := 2;
  C_PRIMARY_METHANE_SENSOR_INDEX : INT := 1;
  C_PRIMARY_EFFECTIVE_GAS_INDEX : INT := 1;
  C_MAX_VENT_UNITS : INT := 8;
  C_MAX_SUPPLY_TEMPS : INT := 2;
  C_MAX_SMOKE_SENSORS : INT := 6;
  C_MAX_SCENARIOS : INT := 6;
  C_MAX_OUTDOOR_ZONES : INT := 4;
  C_MAX_ACCESS_CODES : INT := 10;
  C_MAX_WET_ZONES : INT := 4;
  C_MAX_CALIBRATIONS : INT := 20;
  C_MAX_MODULES : INT := 10;
  C_MAX_CLEANING_MODES : INT := 3;
  C_MAX_ALLOWED_IPS : INT := 5;
  C_MAX_VENT_SUPPLY_MODES : INT := 3;
  C_MAX_SECURITY_PHONES : INT := 5;
  C_MAX_FLOOD_VALVES : INT := 3;
  C_MAX_HUMIDITY_SENSORS : INT := 8;
  C_MAX_CO2_SENSORS : INT := 8;
  C_MAX_CIRCUITS_PER_MANIFOLD : INT := 4;
  C_MAX_TREND_DATA_POINTS : INT := 100;
  C_MAX_HISTORY_RECORDS : INT := 100;
  C_MAX_DEBUG_LOGS : INT := 1000;
  C_MAX_GATEWAY_COMMANDS : INT := 10;
  C_MAX_STATE_SNAPSHOTS : INT := 10;
  C_MAX_BLACKBOX_RECORDS : INT := 100;
  C_MAX_PRESENCE_HISTORY : INT := 1008;
  C_MAX_MODBUS_REGISTERS : INT := 201;
  C_MAX_DEDUPLICATION_HISTORY : INT := 100;
  C_MAX_NVRAM_RECORDS : INT := 100;
  C_MAX_NVRAM_DATA : INT := 128;
  C_MAX_WATER_ZONES : INT := 32;
  C_ANALOG_RAW_MAX : WORD := 27648;
  C_ANALOG_4MA_RAW : WORD := 5529;
  C_ANALOG_3_6MA_RAW : WORD := 4976;
  C_ANALOG_21MA_RAW : WORD := 29030;
  C_ANALOG_10V_MAX_RAW : WORD := 30000;
  C_MS_IN_SECOND : UDINT := 1000;
  C_MS_IN_MINUTE : UDINT := 60000;
  C_MS_IN_HOUR : UDINT := 3600000;
  C_MS_IN_DAY : UDINT := 86400000;
  C_BOILER_CASCADE_MIN_DEMAND : REAL := 25.0;
  C_BOILER_CASCADE_HIGH_DEMAND : REAL := 250.0;
  C_BOILER_SETPOINT_MIN : REAL := 35.0;
  C_BOILER_SETPOINT_MAX : REAL := 55.0;
  C_MIN_HEATING_MANIFOLD_PRESSURE : REAL := 0.8;
END_VAR

VAR_GLOBAL  (* GVL_INTENT_SAFETY *)
  I_Source_Valid : BOOL := FALSE;
  I_Last_Update_Cycle : UDINT := 0;
  I_Last_Update_MS : UDINT := 0;
  I_Fire_Alarm_Active : BOOL := FALSE;
  I_Gas_Alarm_Active : BOOL := FALSE;
  I_Leak_Alarm_Active : BOOL := FALSE;
  I_CO_Warning_Active : BOOL := FALSE;
  I_System_Safe_Stop_Required : BOOL := FALSE;
  I_Freeze_Protection_Required : BOOL := FALSE;
  I_Evacuation_Mode_Active : BOOL := FALSE;
  I_Gas_Close_Required : BOOL := FALSE;
  I_Boiler_Stop_Required : BOOL := FALSE;
  I_Vent_Stop_Required : BOOL := FALSE;
  I_Vent_Force_PV3_Boost : BOOL := FALSE;
  I_Vent_Force_Supply_100 : BOOL := FALSE;
  I_Vent_Force_Supply_80 : BOOL := FALSE;
  I_Vent_Force_Exhaust_100 : BOOL := FALSE;
  I_Water_Main_Close_Required : BOOL := FALSE;
  I_Water_Zone_Close_Required : ARRAY[1..32] OF BOOL;
  I_Water_Selective_Recovery_Allowed : BOOL := FALSE;
  I_Water_Recovery_Target_Zone : INT := 0;
  I_Lock_1_Force_Open : BOOL := FALSE;
  I_Lock_1_Force_Close_Block : BOOL := FALSE;
  I_Lock_2_Force_Open : BOOL := FALSE;
  I_Lock_2_Force_Close_Block : BOOL := FALSE;
  I_Test_Timeout_Gas_Close : BOOL := FALSE;
  I_Test_Timeout_Water_Close : BOOL := FALSE;
END_VAR

{attribute 'qualified_only'}
VAR_GLOBAL  (* GVL_Water_Runtime_Projection *)
  G_Leak_Runtime_State : ARRAY[1..GVL_CONSTANTS.C_MAX_FLOOD_SENSORS] OF ST_Water_Leak_Runtime_State;
  G_Projection_Valid : BOOL;
  G_Last_Projection_MS : UDINT;
  G_Global_Leak_Active : BOOL;
  G_Global_Warning_Active : BOOL;
  G_Runtime_Projection_Status_Code : UINT;
  G_Runtime_Projection_Status_Text : STRING(128);
END_VAR

{attribute 'qualified_only'}
VAR_GLOBAL  (* GVL_Distributed_Runtime *)
  G_Local_Node_State : ST_Distributed_Runtime_Node_State;
  G_Remote_Node_State : ARRAY[1..8] OF ST_Distributed_Runtime_Node_State;
  G_Replication_TX : ARRAY[1..64] OF ST_Distributed_Runtime_Message;
  G_Replication_RX : ARRAY[1..64] OF ST_Distributed_Runtime_Message;
  G_Last_Replication_Sequence_Id : UDINT;
END_VAR

VAR_GLOBAL  (* GVL_POWER_DOMAIN_SEGMENTATION_FABRIC *)
  Power_Domain_Segmentation_Valid : BOOL := FALSE;
  Power_Domain_Segmentation_Granted : BOOL := FALSE;
  Power_Domain_Boundaries_Canonical : BOOL := FALSE;
  Distributed_Power_Segmentation_Stable : BOOL := FALSE;
  Power_Reactivation_Isolation_Valid : BOOL := FALSE;
  Power_Segmentation_Causality_Valid : BOOL := FALSE;
  Power_Recovery_Ordering_Stable : BOOL := FALSE;
  Unsafe_Power_Resurrection_Detected : BOOL := FALSE;
  Partial_Power_Isolation_Asymmetry : BOOL := FALSE;
  Distributed_Power_Segmentation_Fork : BOOL := FALSE;
  Power_Domain_Segmentation_Epoch : UDINT := 0;
END_VAR

{attribute 'qualified_only'}
VAR_GLOBAL  (* GVL_Distributed_Orchestration *)
  G_Topology_Domain : ARRAY[1..32] OF ST_Distributed_Topology_Domain;
  G_Orchestration_State : ST_Distributed_Orchestration_State;
END_VAR

{attribute 'qualified_only'}
VAR_GLOBAL  (* GVL_Water_Hydraulic_Graph *)
  G_Topology_Edge : ARRAY[1..64] OF ST_Water_Hydraulic_Topology_Edge;
  G_Isolation_Path : ARRAY[1..64] OF ST_Water_Isolation_Path_Runtime_State;
  G_Any_Shared_Trunk : BOOL;
  G_Any_Conflict : BOOL;
  G_Any_Global_Fallback_Required : BOOL;
  G_Runtime_Valid : BOOL;
  G_Last_Update_MS : UDINT;
  G_Status_Code : UINT;
  G_Status_Text : STRING(128);
END_VAR

{attribute 'qualified_only'}
VAR_GLOBAL  (* GVL_HEALTH_BRIDGE *)
  G_Smoke_Detected : BOOL;
  G_Gas_Detected : BOOL;
  G_Leak_Detected : BOOL;
  G_Leak_Warning_Level : BOOL;
  G_CO_Warning_Level : BOOL;
  G_CO_Alarm_Level : BOOL;
  G_Last_Fault_Event_Text : STRING(255);
  G_Role_Conflict_Error : BOOL;
END_VAR

{attribute 'qualified_only'}
VAR_GLOBAL  (* GVL_HEATING_POLICY *)
  G_Zone_Empty_Duration_MS : ARRAY[1..GVL_CONSTANTS.C_MAX_ZONES] OF UDINT;
  G_Zone_Permanent_Use : ARRAY[1..GVL_CONSTANTS.C_MAX_ZONES] OF BOOL;
  G_Zone_Guest_Preheat_Request : ARRAY[1..GVL_CONSTANTS.C_MAX_ZONES] OF BOOL;
  G_Zone_Policy_Class : ARRAY[1..GVL_CONSTANTS.C_MAX_ZONES] OF INT;
  G_Zone_Target_Adjustment : ARRAY[1..GVL_CONSTANTS.C_MAX_ZONES] OF REAL;
  G_Zone_Priority_Bias : ARRAY[1..GVL_CONSTANTS.C_MAX_ZONES] OF REAL;
  G_Policy_Mode : E_Heating_Policy_Mode := E_Heating_Policy_Mode.HPM_NORMAL;
  G_Policy_Block_Heating_Request : BOOL;
  G_Policy_Target_Adjustment : REAL;
  G_Policy_Priority_Multiplier : REAL := 1.0;
  G_Policy_Self_Tune_Active : BOOL;
  G_Policy_Self_Tune_Level : INT;
  G_Policy_Feedback_Stable : BOOL;
  G_Policy_Feedback_Improving : BOOL;
  G_Policy_Feedback_Quality : REAL;
  G_Policy_Predictive_Active : BOOL;
  G_Policy_Predictive_Adjustment : REAL;
  G_Zone_Quality : ARRAY[1..GVL_CONSTANTS.C_MAX_ZONES] OF REAL;
  G_Zone_Improving : ARRAY[1..GVL_CONSTANTS.C_MAX_ZONES] OF BOOL;
  G_Zone_Stable : ARRAY[1..GVL_CONSTANTS.C_MAX_ZONES] OF BOOL;
  G_Zone_Self_Level : ARRAY[1..GVL_CONSTANTS.C_MAX_ZONES] OF INT;
  G_Zone_Thermal_Inertia : ARRAY[1..GVL_CONSTANTS.C_MAX_ZONES] OF REAL := [1.0, 1.0, 1.0, 1.0, 1.0, 1.0, 1.0, 1.0, 1.0, 1.0, 1.0, 1.0, 1.0, 1.0, 1.0, 1.0];
  G_Zone_Thermal_Response : ARRAY[1..GVL_CONSTANTS.C_MAX_ZONES] OF REAL;
  G_Zone_Thermal_Demand : ARRAY[1..GVL_CONSTANTS.C_MAX_ZONES] OF REAL;
  G_Zone_Time_To_Heat_MS : ARRAY[1..GVL_CONSTANTS.C_MAX_ZONES] OF UDINT;
  G_Zone_Preheat_Needed : ARRAY[1..GVL_CONSTANTS.C_MAX_ZONES] OF BOOL;
  G_Zone_Heat_Loss_Rate : ARRAY[1..GVL_CONSTANTS.C_MAX_ZONES] OF REAL;
  G_Zone_Heat_Gain_Rate : ARRAY[1..GVL_CONSTANTS.C_MAX_ZONES] OF REAL;
  G_Zone_Predicted_Temp_30m : ARRAY[1..GVL_CONSTANTS.C_MAX_ZONES] OF REAL;
  G_Zone_Thermal_Model_Confidence : ARRAY[1..GVL_CONSTANTS.C_MAX_ZONES] OF REAL;
  G_Zone_Optimization_Score : ARRAY[1..GVL_CONSTANTS.C_MAX_ZONES] OF REAL;
  G_Optimization_Load_Index : REAL;
  G_Optimization_Energy_Saving_Active : BOOL;
  G_Zone_Schedule_Enabled : ARRAY[1..GVL_CONSTANTS.C_MAX_ZONES] OF BOOL;
  G_Zone_Comfort_Time_MS : ARRAY[1..GVL_CONSTANTS.C_MAX_ZONES] OF UDINT;
  G_Zone_Schedule_Preheat_Active : ARRAY[1..GVL_CONSTANTS.C_MAX_ZONES] OF BOOL;
  G_Zone_Schedule_Learned_Offset_MS : ARRAY[1..GVL_CONSTANTS.C_MAX_ZONES, 1..3] OF UDINT;
END_VAR

VAR_GLOBAL  (* GVL_GOVERNANCE_FEEDBACK_INTEGRITY_FABRIC *)
  Governance_Feedback_Integrity_Valid : BOOL := FALSE;
  Governance_Feedback_Integrity_Granted : BOOL := FALSE;
  Governance_Feedback_Integrity_Quarantine_Active : BOOL := TRUE;
  Execution_Feedback_Causality_Isolated : BOOL := FALSE;
  Governance_Derivation_Inputs_Canonical : BOOL := FALSE;
  Telemetry_To_Authority_Lineage_Valid : BOOL := FALSE;
  Feedback_Epoch_Integrity_Stable : BOOL := FALSE;
  Governance_Feedback_Lineage_Coherent : BOOL := FALSE;
  Authenticated_Execution_Observation_Valid : BOOL := FALSE;
  CrossEpoch_Feedback_Continuity_Stable : BOOL := FALSE;
  Governance_Input_Causality_Grounded : BOOL := FALSE;
  Distributed_Feedback_Consensus_Valid : BOOL := FALSE;
  Governance_Feedback_Poisoning_Detected : BOOL := FALSE;
  Execution_Telemetry_Authority_Corruption : BOOL := FALSE;
  CrossEpoch_Feedback_Lineage_Drift : BOOL := FALSE;
  Retroactive_Governance_Mutation_Detected : BOOL := FALSE;
  Distributed_Feedback_Fork_Detected : BOOL := FALSE;
  Untrusted_Execution_Observation_Injected : BOOL := FALSE;
  Governance_Feedback_Integrity_Epoch : UDINT := 0;
  Governance_Feedback_Integrity_Epoch_Coherent : BOOL := FALSE;
  Governance_Feedback_Integrity_Last_Update_MS : UDINT := 0;
  Governance_Feedback_Integrity_Lease_Expired : BOOL := TRUE;
  Governance_Feedback_Integrity_Last_Error_Code : UDINT := 0;
  Governance_Feedback_Integrity_Last_Error_Text : STRING(160) := '';
  Governance_Feedback_Integrity_Invalidation_Count : UDINT := 0;
END_VAR

VAR_GLOBAL  (* GVL_AUTHORITY_RESTORATION *)
  Authority_Restoration_Active : BOOL := FALSE;
  Authority_Restoration_Allowed : BOOL := FALSE;
  Authority_Restoration_Completed : BOOL := FALSE;
  Snapshot_Restoration_Valid : BOOL := FALSE;
  Consensus_Restoration_Valid : BOOL := FALSE;
  Causality_Restoration_Valid : BOOL := FALSE;
  Epoch_Restoration_Valid : BOOL := FALSE;
  Lineage_Restoration_Valid : BOOL := FALSE;
  Revocation_Clearance_Valid : BOOL := FALSE;
  Stabilization_Window_Elapsed : BOOL := FALSE;
  Reauthorization_Order_Valid : BOOL := FALSE;
  Premature_Restoration_Detected : BOOL := FALSE;
  Partial_Restoration_Detected : BOOL := FALSE;
  Restoration_Replay_Suspected : BOOL := FALSE;
  Quarantine_Exit_Race_Detected : BOOL := FALSE;
  Restoration_Epoch : UDINT := 0;
  Restoration_Last_Update_MS : UDINT := 0;
  Restoration_Last_Error_Code : UDINT := 0;
  Restoration_Last_Error_Text : STRING(160) := '';
  Restoration_Invalidation_Count : UDINT := 0;
END_VAR

VAR_GLOBAL  (* GVL_CONVERGENCE *)
  Recovery_Stable_Cycle_Count : UDINT := 0;
  Recovery_Stable_Time_MS : UDINT := 0;
  Convergence_Healthy_Observed : BOOL := FALSE;
  Convergence_Lease_OK : BOOL := FALSE;
  Convergence_Release_Allowed : BOOL := FALSE;
  Convergence_Oscillation_Quarantine_Active : BOOL := FALSE;
  Convergence_Last_Healthy_MS : UDINT := 0;
  Convergence_Last_Invalidation_MS : UDINT := 0;
  Convergence_Invalidation_Count : UDINT := 0;
  Convergence_Min_Stable_Cycles : UDINT := 5;
  Convergence_Min_Stable_Time_MS : UDINT := 500;
  Convergence_Runtime_Barrier_OK : BOOL := FALSE;
  Convergence_Runtime_Snapshot_OK : BOOL := FALSE;
  Convergence_Distributed_Snapshot_OK : BOOL := FALSE;
  Convergence_Distributed_Commit_OK : BOOL := FALSE;
  Convergence_Semantic_Progress_OK : BOOL := FALSE;
  Convergence_Output_Freshness_OK : BOOL := FALSE;
  Convergence_Last_Error_Code : UDINT := 0;
  Convergence_Last_Error_Text : STRING(160) := '';
END_VAR

VAR_GLOBAL  (* GVL_UNSAFE_TRANSITION_FORENSICS_FABRIC *)
  Unsafe_Transition_Forensics_Valid : BOOL := FALSE;
  Unsafe_Transition_Forensics_Granted : BOOL := FALSE;
  Unsafe_Transition_Lineage_Preserved : BOOL := FALSE;
  Forensic_Causality_Continuity_Valid : BOOL := FALSE;
  Distributed_Unsafe_Event_Consensus : BOOL := FALSE;
  Unsafe_Transition_Timeline_Stable : BOOL := FALSE;
  Historical_Safety_Lineage_Coherent : BOOL := FALSE;
  Unsafe_Transition_Hidden : BOOL := FALSE;
  Forensic_Lineage_Break_Detected : BOOL := FALSE;
  Historical_Safety_Gap_Detected : BOOL := FALSE;
  Unsafe_Transition_Forensics_Epoch : UDINT := 0;
END_VAR

{attribute 'qualified_only'}
VAR_GLOBAL  (* GVL_Water_Runtime_Hardening *)
  G_Recovery_FSM : ARRAY[1..64] OF ST_Water_Recovery_FSM_State;
  G_Event_Log : ARRAY[1..128] OF ST_Water_Event_Log_Record;
  G_Runtime_Quarantine_Active : BOOL;
  G_Service_Mode_Active : BOOL;
  G_Maintenance_Mode_Active : BOOL;
  G_Any_Rollback_Required : BOOL;
  G_Any_Escalation_Required : BOOL;
  G_Runtime_Valid : BOOL;
  G_Last_Update_MS : UDINT;
  G_Status_Code : UINT;
  G_Status_Text : STRING(128);
END_VAR

{attribute 'qualified_only'}
VAR_GLOBAL  (* GVL_Water_Isolation_Runtime *)
  G_Isolation_Runtime_State : ARRAY[1..GVL_CONSTANTS.C_MAX_FLOOD_SENSORS] OF ST_Water_Isolation_Runtime_State;
  G_Any_Isolation_Requested : BOOL;
  G_Any_Selective_Isolation : BOOL;
  G_Global_Fallback_Required : BOOL;
  G_Runtime_Valid : BOOL;
  G_Last_Update_MS : UDINT;
  G_Status_Code : UINT;
  G_Status_Text : STRING(128);
END_VAR

VAR_GLOBAL  (* GVL_POLICY *)
  G_Rule_Preheat_Request : BOOL := FALSE;
  G_Scenario_Request_Operator : E_SCENARIO_TYPE := E_SCENARIO_TYPE.SCENARIO_NONE;
  G_Scenario_Request_Gateway : E_SCENARIO_TYPE := E_SCENARIO_TYPE.SCENARIO_NONE;
  G_Scenario_Request_Rule : E_SCENARIO_TYPE := E_SCENARIO_TYPE.SCENARIO_NONE;
  G_Scenario_Intent : E_SCENARIO_TYPE := E_SCENARIO_TYPE.SCENARIO_NONE;
  G_Scenario_Source : E_SCENARIO_SOURCE := SRC_NONE;
END_VAR

FUNCTION_BLOCK FB_IO_Module_Watchdog
  VAR_INPUT
    VI_System_Time_MS : UDINT;
    VI_Module_ID : BYTE;
    VI_Heartbeat_Signal : BOOL;
    VI_Timeout_MS : UDINT := 2000;
  END_VAR
  VAR_OUTPUT
    VO_Module_Online : BOOL;
    VO_Error_Active : BOOL;
  END_VAR
  VAR
    L_Last_Heartbeat_State : BOOL;
    L_Last_Heartbeat_Time : UDINT;
    L_Elapsed_Time : UDINT;
  END_VAR

            // Отслеживание изменения сигнала
IF VI_Heartbeat_Signal <> L_Last_Heartbeat_State THEN
    L_Last_Heartbeat_Time := VI_System_Time_MS;
    L_Last_Heartbeat_State := VI_Heartbeat_Signal;
END_IF;

// Проверка таймаута
L_Elapsed_Time := (SEL(VI_System_Time_MS >= L_Last_Heartbeat_Time, VI_System_Time_MS - L_Last_Heartbeat_Time, (4294967295 - L_Last_Heartbeat_Time) + VI_System_Time_MS + 1));

IF L_Elapsed_Time > VI_Timeout_MS THEN
    VO_Module_Online := FALSE;
    VO_Error_Active := TRUE;
ELSE
    VO_Module_Online := TRUE;
    VO_Error_Active := FALSE;
END_IF;
// >>> BULK_SYNC_ANCHOR: FB_IO_Module_Watchdog <<<
          
END_FUNCTION_BLOCK

FUNCTION_BLOCK FB_HMI_Config_Workflow_Runtime
  VAR_INPUT
    VI_Enable : BOOL;
    VI_System_Time_MS : UDINT;
  END_VAR
  VAR
    L_State : ST_HMI_Config_Workflow_State;
  END_VAR

            IF NOT VI_Enable THEN
    GVL_HMI_Config_Workflow.G_Runtime_Valid := FALSE;
    RETURN;
END_IF;

L_State.Runtime_Valid := TRUE;
L_State.Runtime_System_Time_MS := VI_System_Time_MS;

L_State.Editor_Open :=
    GVL_HMI_Config_Workflow.G_Open_Editor_Request;

L_State.Validation_Requested :=
    GVL_HMI_Config_Workflow.G_Validate_Request;

L_State.Activation_Requested :=
    GVL_HMI_Config_Workflow.G_Activate_Request;

L_State.Rollback_Requested :=
    GVL_HMI_Config_Workflow.G_Rollback_Request;

L_State.Active_Version :=
    GVL_Water_Topology_Config.G_Active_Config_Version;

L_State.Draft_Version :=
    GVL_Config_Activation.G_Staged_Config_Version;

L_State.Last_Stable_Version :=
    GVL_Config_Activation.G_Last_Stable_Config_Version;

L_State.Quarantine_Visible :=
    GVL_Config_Activation.G_Config_Quarantine_Active;

L_State.Service_Mode_Required := TRUE;
L_State.Operator_Ack_Required := TRUE;

IF L_State.Editor_Open THEN
    L_State.Edit_Session_Active := TRUE;
END_IF;

IF L_State.Validation_Requested THEN

    IF GVL_Config_Activation.G_Activation_State.Staged_Config_Valid THEN

        L_State.Validation_OK := TRUE;

    ELSE

        L_State.Validation_Failed := TRUE;

    END_IF;

END_IF;

IF L_State.Activation_Requested THEN

    IF GVL_HMI_Config_Workflow.G_Service_Mode_Active
       AND GVL_HMI_Config_Workflow.G_Operator_Ack
       AND L_State.Validation_OK THEN

        L_State.Activation_Allowed := TRUE;
        GVL_Config_Activation.G_Activation_Request := TRUE;

    ELSE

        L_State.Activation_Blocked := TRUE;

    END_IF;

END_IF;

IF L_State.Rollback_Requested THEN

    IF GVL_HMI_Config_Workflow.G_Operator_Ack THEN

        L_State.Rollback_Allowed := TRUE;
        GVL_Config_Activation.G_Rollback_Request := TRUE;

    END_IF;

END_IF;

IF L_State.Activation_Blocked THEN

    L_State.Status_Code := 2;
    L_State.Status_Text := 'HMI activation blocked';

ELSIF L_State.Validation_Failed THEN

    L_State.Status_Code := 1;
    L_State.Status_Text := 'HMI validation failed';

ELSE

    L_State.Status_Code := 0;
    L_State.Status_Text := 'HMI config workflow healthy';

END_IF;

GVL_HMI_Config_Workflow.G_Workflow_State := L_State;

GVL_HMI_Config_Workflow.G_Runtime_Valid := TRUE;
GVL_HMI_Config_Workflow.G_Last_Update_MS := VI_System_Time_MS;
GVL_HMI_Config_Workflow.G_Status_Code := L_State.Status_Code;
GVL_HMI_Config_Workflow.G_Status_Text := L_State.Status_Text;
          
END_FUNCTION_BLOCK

FUNCTION_BLOCK FB_FloorHeating_Controller
  VAR_INPUT
    VI_Current_Temp : REAL;
    VI_Config : ST_FloorHeating_Circuit_Config;
    VI_Tariff : ST_Tariff_Config;
    VI_Current_Hour : UINT;
    VI_IsActivePLC : BOOL;
    VI_System_Time_MS : UDINT;
  END_VAR
  VAR_OUTPUT
    VO_Pump_Run : BOOL;
    VO_Valve_Pos : REAL;
    VO_Valve_Bool : BOOL;
    VO_Effective_Setpoint : REAL;
  END_VAR
  VAR
    L_Is_Night : BOOL;
    L_PID : FB_PID_Controller;
    L_Last_Time : UDINT;
    L_Cycle_Time_S : REAL;
    L_PWM_Period_MS : UDINT;
    L_PWM_Duty_MS : UDINT;
    L_Current_Phase_MS : UDINT;
    L_PWM_Start_Time : UDINT;
  END_VAR

            // Вычисление времени цикла
IF L_Last_Time = 0 THEN
    L_Last_Time := VI_System_Time_MS;
    L_Cycle_Time_S := 1.0;
ELSE
    L_Cycle_Time_S := UDINT_TO_REAL((SEL(VI_System_Time_MS >= L_Last_Time, VI_System_Time_MS - L_Last_Time, (4294967295 - L_Last_Time) + VI_System_Time_MS + 1))) / 1000.0;
    L_Last_Time := VI_System_Time_MS;
END_IF;
IF L_Cycle_Time_S <= 0.0 THEN L_Cycle_Time_S := 0.01; END_IF;

// 1. Определение активного тарифа
IF VI_Tariff.Enabled THEN
    IF VI_Tariff.Night_Start_Hour > VI_Tariff.Night_End_Hour THEN
        // Переход через полночь (например, 23:00 - 07:00)
        L_Is_Night := (VI_Current_Hour >= VI_Tariff.Night_Start_Hour) OR (VI_Current_Hour < VI_Tariff.Night_End_Hour);
    ELSE
        // В пределах одного дня
        L_Is_Night := (VI_Current_Hour >= VI_Tariff.Night_Start_Hour) AND (VI_Current_Hour < VI_Tariff.Night_End_Hour);
    END_IF;
ELSE
    L_Is_Night := FALSE;
END_IF;

// 2. Расчет эффективной уставки
VO_Effective_Setpoint := VI_Config.design_temp;
IF L_Is_Night THEN
    VO_Effective_Setpoint := VO_Effective_Setpoint + VI_Tariff.Boost_Delta;
END_IF;

// 3. ПИД-регулирование
L_PID(
    VI_SetPoint := VO_Effective_Setpoint,
    VI_ProcessValue := VI_Current_Temp,
    VI_Kp := VI_Config.pid_kp,
    VI_Tn := 300.0,
    VI_Tv := 0.0,
    VI_Y_Min := 0.0,
    VI_Y_Max := 100.0,
    VI_Cycle_Time_S := L_Cycle_Time_S,
    VO_Output => VO_Valve_Pos
);

// 4. ШИМ-модуляция для термоэлектрического привода
IF VI_Config.pwm_period_s > 0 THEN
    L_PWM_Period_MS := TO_UDINT(VI_Config.pwm_period_s) * 1000;
ELSE
    L_PWM_Period_MS := 600000; // 10 минут
END_IF;

L_Current_Phase_MS := (SEL(VI_System_Time_MS >= L_PWM_Start_Time, VI_System_Time_MS - L_PWM_Start_Time, (4294967295 - L_PWM_Start_Time) + VI_System_Time_MS + 1));
IF L_Current_Phase_MS >= L_PWM_Period_MS THEN
    L_PWM_Start_Time := VI_System_Time_MS - (L_Current_Phase_MS - L_PWM_Period_MS); // Сохраняем остаток для точности
    L_Current_Phase_MS := (SEL(VI_System_Time_MS >= L_PWM_Start_Time, VI_System_Time_MS - L_PWM_Start_Time, (4294967295 - L_PWM_Start_Time) + VI_System_Time_MS + 1));
END_IF;

L_PWM_Duty_MS := TO_UDINT((VO_Valve_Pos / 100.0) * TO_REAL(L_PWM_Period_MS));

IF VI_IsActivePLC THEN
    VO_Pump_Run := (VO_Valve_Pos > 5.0);
    
    IF VO_Valve_Pos >= 100.0 THEN
        VO_Valve_Bool := TRUE;
    ELSIF VO_Valve_Pos <= 0.0 THEN
        VO_Valve_Bool := FALSE;
    ELSE
        VO_Valve_Bool := (L_Current_Phase_MS <= L_PWM_Duty_MS);
    END_IF;
ELSE
    VO_Pump_Run := FALSE;
    VO_Valve_Bool := FALSE;
END_IF;
          
END_FUNCTION_BLOCK

FUNCTION_BLOCK FB_Heating_RootCause_Diagnostics
  VAR_INPUT
    VI_Enable : BOOL;
  END_VAR
  VAR
    fbRootCause : FB_Diagnostics_RootCause;
    fbDemandMap : FB_Heating_Demand_Map;
    L_Demand_Map : ARRAY[1..GVL_CONSTANTS.C_MAX_MANIFOLDS] OF BOOL;
  END_VAR

            // ==============================================================================
// Heating root-cause diagnostics observer
// Public diagnostics/explainability layer.
// Does NOT own control/runtime decisions.
// ==============================================================================



IF NOT VI_Enable THEN
    GVL_STATE.G_Heating_RootCause := E_Heating_RootCause.RC_NONE;
    GVL_STATE.G_Heating_RootConfidence := 0.0;
    GVL_STATE.G_Heating_Confidence := 0.0;
    GVL_STATE.G_Heating_Error_Score := 1.0;
    GVL_STATE.G_Heating_Confidence_Reason_Code := -1;
    GVL_STATE.G_Heating_Confidence_Reason_Text := 'Heating diagnostics disabled';
    RETURN;
END_IF;

// ======================================================
// DEMAND MAP
// ======================================================
fbDemandMap(
    VI_Zone_Valves := GVL_STATE.G_Zone_Valves,
    VI_Zone_Configs := GVL_CONFIG.G_HMI_FloorHeating_Configs,
    VO_Manifold_Demand_Map => L_Demand_Map
);

// ======================================================
// INTERNAL INFERENCE ENGINE
// ======================================================
fbRootCause(
    VI_Emergency_Stop := GVL_STATE.G_Safety_Emergency_Stop,
    VI_Gas_Safety := GVL_STATE.G_Safety_Gas_Latched,
    VI_IO_Failsafe := GVL_STATE.G_Heating_IO_Fault,

    VI_Cascade_Available := GVL_STATE.G_Heating_Cascade_Available,
    VI_Cascade_Degraded := GVL_STATE.G_Heating_Cascade_Degraded,
    VI_Cascade_Partial_Capacity := GVL_STATE.G_Heating_Cascade_Partial_Capacity,
    VI_Cascade_No_Flame := GVL_STATE.G_Heating_Cascade_No_Flame,
    VI_Cascade_Transport_Degraded := GVL_STATE.G_Heating_Cascade_Transport_Degraded,
    VI_Cascade_Ignition_Timeout := GVL_STATE.G_Heating_Cascade_Ignition_Timeout,
    VI_Cascade_Active_Boilers := GVL_STATE.G_Heating_Cascade_Active_Boilers,
    VI_Cascade_Available_Boilers := GVL_STATE.G_Heating_Cascade_Available_Boilers,

    VI_Boiler_OT_Online := GVL_STATE.G_Boiler_OT_Online,
    VI_Boiler_Error := GVL_STATE.G_Boiler_Error,
    VI_Boiler_Flame := GVL_STATE.G_Boiler_Flame,
    VI_Boiler_OT_Command_Timeout := GVL_STATE.G_Boiler_OT_Command_Timeout,
    VI_Boiler_OT_Heartbeat_Timeout := GVL_STATE.G_Boiler_OT_Heartbeat_Timeout,
    VI_Boiler_OT_Adapter_Error := GVL_STATE.G_Boiler_OT_Adapter_Error,

    VI_Manifold_Pumps := GVL_STATE.G_Manifold_Pumps,
    VI_Manifold_Valves := GVL_STATE.G_Manifold_Valves,

    VI_Sensor_Error := GVL_STATE.G_Heating_Sensor_Fault,
    VI_Supply_Temps := GVL_STATE.G_Manifold_T_Supply,
    VI_Target_Supply := GVL_STATE.G_Target_Temperature,
    VI_Demand_Map := L_Demand_Map
);

// ======================================================
// PUBLIC DIAGNOSTICS STATE
// ======================================================
GVL_STATE.G_Heating_RootCause := fbRootCause.VO_RootCause;
GVL_STATE.G_Heating_RootConfidence := fbRootCause.VO_Confidence;
GVL_STATE.G_Heating_Confidence := fbRootCause.VO_Confidence;
GVL_STATE.G_Heating_Error_Score := fbRootCause.VO_Error_Score;
GVL_STATE.G_Heating_Confidence_Reason_Code := fbRootCause.VO_Reason_Code;
GVL_STATE.G_Heating_Confidence_Reason_Text := fbRootCause.VO_Reason_Text;

// >>> BULK_SYNC_ANCHOR: FB_Heating_RootCause_Diagnostics <<<
          
END_FUNCTION_BLOCK

FUNCTION_BLOCK FB_State_Trace_Log
  VAR_INPUT
    VI_System_Time : UDINT;
    VI_Gas_Alarm : BOOL;
    VI_Leak_Alarm : BOOL;
    VI_Pumps : ARRAY[1..4] OF BOOL;
  END_VAR
  VAR_OUTPUT
    VO_Last_Change_Time : UDINT;
  END_VAR
  VAR
    L_Last_Gas : BOOL;
    L_Last_Leak : BOOL;
  END_VAR

            IF (VI_Gas_Alarm <> L_Last_Gas) OR (VI_Leak_Alarm <> L_Last_Leak) THEN
    VO_Last_Change_Time := VI_System_Time;
END_IF;

L_Last_Gas := VI_Gas_Alarm;
L_Last_Leak := VI_Leak_Alarm;
          
END_FUNCTION_BLOCK

FUNCTION_BLOCK FB_System_Evacuation
  VAR
    L_i : INT;
  END_VAR

            // ==============================================================================
// System evacuation helper
//
// Internal helper for PRG_System.
// Owns evacuation guidance, target/hazard zone name projection,
// and evacuation lighting activation.
// ==============================================================================



FOR L_i := 1 TO 32 DO
    GVL_STATE.G_Evac_Guidance[L_i] := 0;

    IF GVL_STATE.G_Evac_Hazard_Zone[L_i] THEN
        GVL_STATE.G_Evac_Guidance[L_i] := -1;
    END_IF;

    IF GVL_CONFIG.G_Evac_Exit_Zones[L_i] AND NOT GVL_STATE.G_Evac_Hazard_Zone[L_i] THEN
        GVL_STATE.G_Evac_Guidance[L_i] := 1;
    END_IF;
END_FOR;

GVL_STATUS.G_Evac_Target_Zone_Name := '';
GVL_STATUS.G_Evac_Hazard_Zone_Name := '';

FOR L_i := 1 TO 32 DO
    IF (GVL_STATUS.G_Evac_Hazard_Zone_Name = '') AND GVL_STATE.G_Evac_Hazard_Zone[L_i] THEN
        GVL_STATUS.G_Evac_Hazard_Zone_Name := GVL_CONFIG.G_Evac_Zone_Names[L_i];
        IF GVL_STATUS.G_Evac_Hazard_Zone_Name = '' THEN
            GVL_STATUS.G_Evac_Hazard_Zone_Name := CONCAT('Zone ', INT_TO_STRING(L_i));
        END_IF;
    END_IF;

    IF (GVL_STATUS.G_Evac_Target_Zone_Name = '') AND (GVL_STATE.G_Evac_Guidance[L_i] = 1) THEN
        GVL_STATUS.G_Evac_Target_Zone_Name := GVL_CONFIG.G_Evac_Zone_Names[L_i];
        IF GVL_STATUS.G_Evac_Target_Zone_Name = '' THEN
            GVL_STATUS.G_Evac_Target_Zone_Name := CONCAT('Zone ', INT_TO_STRING(L_i));
        END_IF;
    END_IF;
END_FOR;

IF GVL_STATE.G_System_Mode = E_System_Operating_Mode.MODE_SAFE_STOP AND GVL_STATE.G_Safety_Smoke_Latched THEN
    GVL_STATE.G_Evacuation_Lighting_Active := TRUE;
ELSE
    GVL_STATE.G_Evacuation_Lighting_Active := FALSE;
END_IF;

// >>> BULK_SYNC_ANCHOR: FB_System_Evacuation <<<
          
END_FUNCTION_BLOCK

FUNCTION_BLOCK FB_Heating_Runtime_Observer_Authorization
  VAR_INPUT
    VI_Enable_Request : BOOL;
    VI_Bootstrap_Mode : BOOL;
    VI_Passive_Mode : BOOL;
    VI_ReadOnly_Mode : BOOL;
    VI_Governance_Locked : BOOL;
    VI_Runtime_Authority_Disabled : BOOL;
    VI_Writable_Exports_Disabled : BOOL;
  END_VAR
  VAR_OUTPUT
    VO_Enable_Authorized : BOOL;
    VO_Enable_Effective : BOOL;
    VO_Authorization_Valid : BOOL;
    VO_Status_Code : UINT;
    VO_Status_Text : STRING(128);
  END_VAR

            // ==============================================================================
// Heating runtime observer authorization
// Governed passive-bootstrap authorization only.
// Read-only.
// Deterministic.
// ==============================================================================



// ======================================================
// DEFAULTS
// ======================================================
VO_Enable_Authorized := FALSE;
VO_Enable_Effective := FALSE;
VO_Authorization_Valid := FALSE;

VO_Status_Code := 0;
VO_Status_Text := 'Heating runtime observer authorization inactive';

// ======================================================
// REQUEST VALIDATION
// ======================================================
IF NOT VI_Enable_Request THEN
    RETURN;
END_IF;

// ======================================================
// GOVERNANCE VALIDATION
// ======================================================
IF NOT VI_Bootstrap_Mode THEN
    VO_Status_Code := 100;
    VO_Status_Text := 'Bootstrap mode required for observer authorization';
    RETURN;
END_IF;

IF NOT VI_Passive_Mode THEN
    VO_Status_Code := 110;
    VO_Status_Text := 'Passive mode required for observer authorization';
    RETURN;
END_IF;

IF NOT VI_ReadOnly_Mode THEN
    VO_Status_Code := 120;
    VO_Status_Text := 'Read-only mode required for observer authorization';
    RETURN;
END_IF;

IF NOT VI_Governance_Locked THEN
    VO_Status_Code := 130;
    VO_Status_Text := 'Governance lock required for observer authorization';
    RETURN;
END_IF;

IF NOT VI_Runtime_Authority_Disabled THEN
    VO_Status_Code := 140;
    VO_Status_Text := 'Runtime authority isolation required';
    RETURN;
END_IF;

IF NOT VI_Writable_Exports_Disabled THEN
    VO_Status_Code := 150;
    VO_Status_Text := 'Writable exports must remain disabled';
    RETURN;
END_IF;

// ======================================================
// AUTHORIZED PASSIVE BOOTSTRAP ACTIVATION
// ======================================================
VO_Enable_Authorized := TRUE;
VO_Enable_Effective := TRUE;
VO_Authorization_Valid := TRUE;

VO_Status_Code := 1;
VO_Status_Text := 'Heating runtime observer authorization granted';

// >>> BULK_SYNC_ANCHOR: FB_Heating_Runtime_Observer_Authorization <<<
          
END_FUNCTION_BLOCK

FUNCTION_BLOCK FB_HMI_Interface
  VAR_INPUT
    VI_Severity : E_System_Severity;
    VI_RootCause : E_System_Root_Cause;
    VI_Status_Msg : STRING(200);
  END_VAR
  VAR_OUTPUT
    VO_HMI_Status_Text : STRING(200);
    VO_HMI_State_Code : INT;
  END_VAR

            VO_HMI_Status_Text := VI_Status_Msg;

CASE VI_Severity OF
    E_System_Severity.SEV_NORMAL:
        VO_HMI_State_Code := 0;
    E_System_Severity.SEV_WARNING:
        VO_HMI_State_Code := 1;
    E_System_Severity.SEV_DEGRADED:
        VO_HMI_State_Code := 2;
    E_System_Severity.SEV_CRITICAL:
        VO_HMI_State_Code := 3;
ELSE
        // No fallback required
END_CASE;
// >>> BULK_SYNC_ANCHOR: FB_HMI_Interface <<<
          
END_FUNCTION_BLOCK

FUNCTION_BLOCK FB_Time_Service
  VAR
    L_Real_Now : UDINT;
    L_Elapsed : UDINT;
    L_Scaled_Delta : UDINT;
  END_VAR

            // read real time
L_Real_Now := GVL_STATUS.G_System_Time_MS;

// wrap-safe delta (real time base)
IF L_Real_Now >= GVL_TIME_SERVICE.G_Last_Now_MS THEN
    L_Elapsed := L_Real_Now - GVL_TIME_SERVICE.G_Last_Now_MS;
    GVL_TIME_SERVICE.G_Wrap_Detected := FALSE;
ELSE
    L_Elapsed := (16#FFFFFFFF - GVL_TIME_SERVICE.G_Last_Now_MS) + L_Real_Now + 1;
    GVL_TIME_SERVICE.G_Wrap_Detected := TRUE;
END_IF;

GVL_TIME_SERVICE.G_Last_Now_MS := L_Real_Now;

// --- SIMULATION MODE ---
IF GVL_TIME_SERVICE.G_Sim_Enabled THEN

    IF NOT GVL_TIME_SERVICE.G_Sim_Frozen THEN
        L_Scaled_Delta := REAL_TO_UDINT(TO_REAL(L_Elapsed) * GVL_TIME_SERVICE.G_Sim_Time_Scale);

        GVL_TIME_SERVICE.G_Sim_Now_MS := GVL_TIME_SERVICE.G_Sim_Now_MS + L_Scaled_Delta;

        GVL_TIME_SERVICE.G_Sim_Time_Of_Day_MS := GVL_TIME_SERVICE.G_Sim_Time_Of_Day_MS + L_Scaled_Delta;

        IF GVL_TIME_SERVICE.G_Sim_Time_Of_Day_MS >= 86400000 THEN
            GVL_TIME_SERVICE.G_Sim_Time_Of_Day_MS := GVL_TIME_SERVICE.G_Sim_Time_Of_Day_MS MOD 86400000;
            GVL_TIME_SERVICE.G_Sim_Day_Of_Week := GVL_TIME_SERVICE.G_Sim_Day_Of_Week + 1;
            IF GVL_TIME_SERVICE.G_Sim_Day_Of_Week > 7 THEN
                GVL_TIME_SERVICE.G_Sim_Day_Of_Week := 1;
            END_IF;
        END_IF;
    END_IF;

    GVL_TIME_SERVICE.G_Now_MS := GVL_TIME_SERVICE.G_Sim_Now_MS;
    GVL_TIME_SERVICE.G_Time_Of_Day_MS := GVL_TIME_SERVICE.G_Sim_Time_Of_Day_MS;
    GVL_TIME_SERVICE.G_Day_Of_Week := GVL_TIME_SERVICE.G_Sim_Day_Of_Week;

ELSE
    GVL_TIME_SERVICE.G_Now_MS := L_Real_Now;
    GVL_TIME_SERVICE.G_Time_Of_Day_MS := GVL_STATUS.G_Time_Of_Day_MS;
    GVL_TIME_SERVICE.G_Day_Of_Week := TO_INT(GVL_STATUS.G_Current_Day);
END_IF;

// TOD unified
GVL_TIME_SERVICE.G_Current_TOD := UDINT_TO_TOD(GVL_TIME_SERVICE.G_Time_Of_Day_MS);

GVL_TIME_SERVICE.G_Delta_MS := L_Elapsed;
          
END_FUNCTION_BLOCK

FUNCTION_BLOCK FB_Water_Hardware_Binding_Runtime
  VAR_INPUT
    VI_Enable : BOOL;
    VI_System_Time_MS : UDINT;
  END_VAR
  VAR
    L_i : INT;
    L_Channel : UINT;
    L_Binding : ST_IO_Binding_Record;
    L_Any_Invalid : BOOL;
    L_Any_Missing : BOOL;
  END_VAR

            IF NOT VI_Enable THEN
    GVL_IO_Binding_Runtime.G_Runtime_Valid := FALSE;
    RETURN;
END_IF;

FOR L_i := 1 TO GVL_CONSTANTS.C_MAX_FLOOD_SENSORS DO

    // Flood sensor runtime binding.
    L_Binding :=
        GVL_IO_Binding_Config.G_Flood_Sensor_Binding[L_i];

    IF L_Binding.Binding_Valid THEN

        L_Channel := L_Binding.Physical_Channel_Id;

        IF (L_Channel >= 1)
           AND (L_Channel <= GVL_CONSTANTS.C_MAX_FLOOD_SENSORS) THEN

            GVL_IO_Binding_Runtime.G_Flood_Sensor_Value[L_i] :=
                GVL_IO.DI_Flood_Sensors[L_Channel];

            GVL_IO_Binding_Runtime.G_Flood_Sensor_Valid[L_i] := TRUE;

        ELSE

            L_Any_Invalid := TRUE;

        END_IF;

    ELSE

        L_Any_Missing := TRUE;

    END_IF;

    // Valve close feedback runtime binding.
    L_Binding :=
        GVL_IO_Binding_Config.G_Water_Valve_Close_FB_Binding[L_i];

    IF L_Binding.Binding_Valid THEN

        L_Channel := L_Binding.Physical_Channel_Id;

        IF (L_Channel >= 1)
           AND (L_Channel <= GVL_CONSTANTS.C_MAX_WATER_ZONES) THEN

            GVL_IO_Binding_Runtime.G_Water_Valve_Close_FB_Value[L_i] :=
                GVL_IO.DI_Water_Zone_Close_FB[L_Channel];

            GVL_IO_Binding_Runtime.G_Water_Valve_Close_FB_Valid[L_i] := TRUE;

        ELSE

            L_Any_Invalid := TRUE;

        END_IF;

    END_IF;

    // Valve open feedback runtime binding.
    L_Binding :=
        GVL_IO_Binding_Config.G_Water_Valve_Open_FB_Binding[L_i];

    IF L_Binding.Binding_Valid THEN

        L_Channel := L_Binding.Physical_Channel_Id;

        IF (L_Channel >= 1)
           AND (L_Channel <= GVL_CONSTANTS.C_MAX_WATER_ZONES) THEN

            GVL_IO_Binding_Runtime.G_Water_Valve_Open_FB_Value[L_i] :=
                GVL_IO.DI_Water_Zone_Open_FB[L_Channel];

            GVL_IO_Binding_Runtime.G_Water_Valve_Open_FB_Valid[L_i] := TRUE;

        ELSE

            L_Any_Invalid := TRUE;

        END_IF;

    END_IF;

END_FOR;

GVL_IO_Binding_Runtime.G_Any_Invalid_Binding :=
    L_Any_Invalid;

GVL_IO_Binding_Runtime.G_Any_Missing_Binding :=
    L_Any_Missing;

GVL_IO_Binding_Runtime.G_Runtime_Valid := TRUE;
GVL_IO_Binding_Runtime.G_Last_Update_MS := VI_System_Time_MS;

IF L_Any_Invalid THEN
    GVL_IO_Binding_Runtime.G_Status_Code := 2;
    GVL_IO_Binding_Runtime.G_Status_Text :=
        'Hardware binding invalid';
ELSIF L_Any_Missing THEN
    GVL_IO_Binding_Runtime.G_Status_Code := 1;
    GVL_IO_Binding_Runtime.G_Status_Text :=
        'Hardware binding incomplete';
ELSE
    GVL_IO_Binding_Runtime.G_Status_Code := 0;
    GVL_IO_Binding_Runtime.G_Status_Text :=
        'Hardware binding runtime healthy';
END_IF;
          
END_FUNCTION_BLOCK

FUNCTION_BLOCK FB_Heating_Runtime_Meta_Supervision_Publisher
  VAR_INPUT
    VI_Enable : BOOL;
    VI_Runtime_Observation_Valid : BOOL;
    VI_Runtime_Observer_Ready : BOOL;
    VI_Runtime_Observer_Fault : BOOL;
    VI_Runtime_Status_Code : UINT;
    VI_Runtime_Status_Text : STRING(128);
  END_VAR
  VAR_OUTPUT
    VO_Meta : ST_Heating_Runtime_Meta_Supervision;
    VO_Publication_Valid : BOOL;
  END_VAR

            VO_Meta.Meta_Analytics_Visible := FALSE;
VO_Meta.Meta_Analytics_Degraded := FALSE;
VO_Meta.Meta_Analytics_Attention := FALSE;

VO_Meta.Supervision_Integrity_Visible := FALSE;
VO_Meta.Supervision_Integrity_Observation := 0;

VO_Meta.Adaptive_Drift_Visible := FALSE;
VO_Meta.Adaptive_Drift_Observation := 0;

VO_Meta.Confidence_Degradation_Visible := FALSE;
VO_Meta.Confidence_Degradation_Observation := 0;

VO_Meta.Analytics_Consistency_Visible := FALSE;
VO_Meta.Analytics_Consistency_Observation := 0;

VO_Meta.Sequencing_Meta_Observation := FALSE;
VO_Meta.Ownership_Meta_Observation := FALSE;
VO_Meta.Synchronization_Meta_Observation := FALSE;

VO_Meta.Status_Code := 0;
VO_Meta.Status_Text := 'Heating runtime meta supervision inactive';

VO_Publication_Valid := FALSE;

IF NOT VI_Enable THEN
    RETURN;
END_IF;

VO_Meta.Meta_Analytics_Visible := TRUE;
VO_Meta.Supervision_Integrity_Visible := TRUE;
VO_Meta.Adaptive_Drift_Visible := TRUE;
VO_Meta.Confidence_Degradation_Visible := TRUE;
VO_Meta.Analytics_Consistency_Visible := TRUE;

VO_Meta.Sequencing_Meta_Observation := VI_Runtime_Observation_Valid;
VO_Meta.Ownership_Meta_Observation := VI_Runtime_Observer_Ready;
VO_Meta.Synchronization_Meta_Observation := NOT VI_Runtime_Observer_Fault;

IF VI_Runtime_Observer_Fault THEN
    VO_Meta.Meta_Analytics_Degraded := TRUE;
    VO_Meta.Meta_Analytics_Attention := TRUE;
    VO_Meta.Supervision_Integrity_Observation := 900;
ELSIF NOT VI_Runtime_Observation_Valid THEN
    VO_Meta.Meta_Analytics_Attention := TRUE;
    VO_Meta.Supervision_Integrity_Observation := 200;
ELSE
    VO_Meta.Supervision_Integrity_Observation := 1;
END_IF;

VO_Meta.Status_Code := VI_Runtime_Status_Code;
VO_Meta.Status_Text := VI_Runtime_Status_Text;

VO_Publication_Valid := TRUE;

// >>> BULK_SYNC_ANCHOR: FB_Heating_Runtime_Meta_Supervision_Publisher <<<
          
END_FUNCTION_BLOCK

FUNCTION_BLOCK FB_Distributed_Authority_Arbitration
  VAR_INPUT
    VI_Enable : BOOL;
    VI_System_Time_MS : UDINT;
  END_VAR
  VAR
    L_State : ST_Distributed_Authority_State;
    L_Lease_Expired : BOOL;
    L_Finalized_Runtime_Continuity : BOOL;
  END_VAR

            IF NOT VI_Enable THEN
    GVL_Distributed_Authority.G_Runtime_Valid := FALSE;
    RETURN;
END_IF;

L_State.Runtime_Valid := TRUE;
L_State.Runtime_System_Time_MS := VI_System_Time_MS;

L_State.Controller_Id :=
    GVL_Distributed_Runtime.G_Local_Node_State.Controller_Id;

L_State.Runtime_Node_Id :=
    GVL_Distributed_Runtime.G_Local_Node_State.Runtime_Node_Id;

L_State.Authority_Domain_Id :=
    GVL_Distributed_Runtime.G_Local_Node_State.Authority_Domain_Id;

L_State.Authority_Election_Active := TRUE;

L_Lease_Expired :=
    (VI_System_Time_MS - GVL_Distributed_Authority.G_Authority_Lease_Start_MS)
    > GVL_Distributed_Authority.G_Authority_Lease_Duration_MS;

L_State.Authority_Lease_Expired := L_Lease_Expired;
L_State.Authority_Lease_Valid := NOT L_Lease_Expired;

L_State.Replication_Consensus_Healthy :=
    GVL_Distributed_Runtime.G_Distributed_Replication_Healthy;

L_State.Replication_Consensus_Stale :=
    NOT GVL_Distributed_Runtime.G_Distributed_Replication_Healthy;

L_Finalized_Runtime_Continuity :=
    GVL_SEMANTIC_PROGRESS.Semantic_Forward_Progress_Valid
    AND GVL_SEMANTIC_PROGRESS.Semantic_Execution_Continuity_OK
    AND NOT GVL_SEMANTIC_PROGRESS.Semantic_Progress_Lease_Expired
    AND NOT GVL_SEMANTIC_PROGRESS.Semantic_Progress_Quarantine_Active
    AND GVL_RUNTIME_SNAPSHOT.Snapshot_Frozen
    AND GVL_RUNTIME_SNAPSHOT.Snapshot_Publication_Allowed
    AND GVL_RUNTIME_SNAPSHOT.Snapshot_Copy_Valid
    AND GVL_RUNTIME_SNAPSHOT.Snapshot_Isolation_Valid
    AND NOT GVL_RUNTIME_SNAPSHOT.Snapshot_Mutation_Detected
    AND GVL_DISTRIBUTED_SNAPSHOT.Distributed_Publication_Reconciled
    AND GVL_DISTRIBUTED_SNAPSHOT.Distributed_Publication_Freeze_Valid
    AND GVL_DISTRIBUTED_SNAPSHOT.Distributed_Snapshot_Consistent
    AND GVL_DISTRIBUTED_COMMIT.Distributed_Commit_Valid
    AND GVL_DISTRIBUTED_COMMIT.Publication_Prepare_Valid
    AND GVL_DISTRIBUTED_COMMIT.Publication_Commit_Confirmed
    AND NOT GVL_DISTRIBUTED_COMMIT.Peer_Commit_Mismatch
    AND NOT GVL_DISTRIBUTED_COMMIT.Commit_Lease_Expired
    AND GVL_OUTPUT_EPOCH.Output_Publication_Valid
    AND GVL_OUTPUT_EPOCH.Output_Runtime_Epoch_Valid
    AND NOT GVL_OUTPUT_EPOCH.Output_Lease_Expired
    AND NOT GVL_OUTPUT_EPOCH.Output_Forced_Safe_Decay
    AND GVL_COMMAND_VERIFY.PreOutput_Barrier_OK
    AND NOT GVL_COMMAND_VERIFY.PreOutput_Block_IO;

L_State.Distributed_Safety_Barrier_OK :=
    GVL_Runtime_Restart_Continuity.G_Runtime_Valid
    AND NOT GVL_Config_Activation.G_Config_Quarantine_Active
    AND NOT GVL_Distributed_Runtime.G_Split_Brain_Suspected
    AND GVL_IO_Binding_Runtime.G_Runtime_Valid
    AND L_Finalized_Runtime_Continuity;

IF NOT L_State.Distributed_Safety_Barrier_OK THEN

    L_State.Split_Brain_Blocked := TRUE;
    L_State.Authority_Observer_Only := TRUE;

    L_State.Status_Code := 3;
    L_State.Status_Text :=
        'Distributed authority blocked by safety barrier';

ELSIF L_State.Replication_Consensus_Healthy
   AND NOT L_Lease_Expired
   AND L_Finalized_Runtime_Continuity THEN

    L_State.Authority_Master_Elected := TRUE;

    L_State.Recovery_Authority_Allowed := TRUE;
    L_State.Rollback_Authority_Allowed := TRUE;
    L_State.Quarantine_Authority_Allowed := TRUE;

    L_State.Status_Code := 1;
    L_State.Status_Text :=
        'Distributed master authority active';

ELSE

    L_State.Authority_Backup_Elected := TRUE;

    L_State.Status_Code := 2;
    L_State.Status_Text :=
        'Distributed backup authority active';

END_IF;

GVL_Distributed_Authority.G_Authority_State := L_State;

GVL_Distributed_Authority.G_Split_Brain_Blocked :=
    L_State.Split_Brain_Blocked;

GVL_Distributed_Authority.G_Distributed_Safety_Barrier_OK :=
    L_State.Distributed_Safety_Barrier_OK;

GVL_Distributed_Authority.G_Runtime_Valid := TRUE;
GVL_Distributed_Authority.G_Last_Update_MS := VI_System_Time_MS;
GVL_Distributed_Authority.G_Status_Code := L_State.Status_Code;
GVL_Distributed_Authority.G_Status_Text := L_State.Status_Text;
          
END_FUNCTION_BLOCK

FUNCTION_BLOCK FB_Water_Topology_Config_Runtime
  VAR_INPUT
    VI_Enable : BOOL;
    VI_System_Time_MS : UDINT;
  END_VAR
  VAR
    L_i : INT;
    L_Config : ST_Water_Topology_Config_Record;
    L_Any_Invalid : BOOL;
    L_Any_Multi_Valve : BOOL;
  END_VAR

            IF NOT VI_Enable THEN
    GVL_Water_Topology_Config.G_Runtime_Valid := FALSE;
    RETURN;
END_IF;

FOR L_i := 1 TO GVL_CONSTANTS.C_MAX_FLOOD_SENSORS DO

    L_Config := GVL_Water_Topology_Config_Source.G_Source_Record[L_i];

    IF NOT L_Config.Config_Valid THEN
        L_Config.Config_Valid := TRUE;
        L_Config.Config_Version := 1;
        L_Config.Sensor_Id := TO_UINT(L_i);
        L_Config.Logical_Zone_Id := TO_UINT(L_i);
        L_Config.Hydraulic_Segment_Id := TO_UINT(L_i);
        L_Config.Isolation_Group_Id := TO_UINT(L_i);
        L_Config.Primary_Valve_Group_Id := TO_UINT(L_i);
        L_Config.Fallback_Domain_Id := 1;
        L_Config.Recovery_Domain_Id := 1;

        IF (L_i MOD 4) = 0 THEN
            L_Config.Shared_Trunk := TRUE;
            L_Config.Cross_Zone_Dependency := TRUE;
            L_Config.Multi_Valve_Required := TRUE;
            L_Config.Secondary_Valve_Group_Id := TO_UINT(L_i + 100);
        END_IF;
    END_IF;

    IF L_Config.Primary_Valve_Group_Id = 0 THEN
        L_Config.Config_Valid := FALSE;
        L_Config.Status_Code := 1;
        L_Config.Status_Text := 'Invalid topology config';
    ELSE
        L_Config.Status_Code := 0;
        L_Config.Status_Text := 'Topology config loaded';
    END_IF;

    GVL_Water_Topology_Config.G_Config_Record[L_i] := L_Config;

    L_Any_Invalid := L_Any_Invalid OR NOT L_Config.Config_Valid;
    L_Any_Multi_Valve := L_Any_Multi_Valve OR L_Config.Multi_Valve_Required;

END_FOR;

GVL_Water_Topology_Config.G_Active_Config_Version := GVL_Water_Topology_Config_Source.G_Source_Version;
GVL_Water_Topology_Config.G_Config_Loaded := TRUE;
GVL_Water_Topology_Config.G_Runtime_Remap_Ready := TRUE;
GVL_Water_Topology_Config.G_Any_Invalid_Config := L_Any_Invalid;
GVL_Water_Topology_Config.G_Any_Multi_Valve_Required := L_Any_Multi_Valve;
GVL_Water_Topology_Config.G_Runtime_Valid := TRUE;
GVL_Water_Topology_Config.G_Last_Update_MS := VI_System_Time_MS;

IF L_Any_Invalid THEN
    GVL_Water_Topology_Config.G_Status_Code := 2;
    GVL_Water_Topology_Config.G_Status_Text := 'Topology config invalid';
ELSIF L_Any_Multi_Valve THEN
    GVL_Water_Topology_Config.G_Status_Code := 1;
    GVL_Water_Topology_Config.G_Status_Text := 'Multi-valve topology active';
ELSE
    GVL_Water_Topology_Config.G_Status_Code := 0;
    GVL_Water_Topology_Config.G_Status_Text := 'Topology config runtime healthy';
END_IF;
          
END_FUNCTION_BLOCK

FUNCTION_BLOCK FB_Heating_Runtime_Supervisory_Enrichment
  VAR_INPUT
    VI_Enable : BOOL;
    VI_System_Time_MS : UDINT;
    VI_Runtime_Context : ST_Heating_Runtime_Context;
    VI_Phase_Event : ST_Heating_Runtime_Phase_Event;
    VI_Anomaly : ST_Heating_Runtime_Anomaly;
    VI_Cascade_Boiler_Count : UINT;
    VI_OT_Command_Valid : BOOL;
  END_VAR
  VAR_OUTPUT
    VO_Causality_Node : ST_Heating_Runtime_Causality_Node;
    VO_Causality_Edge : ST_Heating_Runtime_Causality_Edge;
    VO_Blackbox_Event : ST_Heating_Runtime_Blackbox_Event;
    VO_Predictive_State : ST_Heating_Runtime_Predictive_State;
    VO_Status_Code : UINT;
    VO_Status_Text : STRING(128);
  END_VAR
  VAR_IN_OUT
    VIO_Event_Buffer : ST_Heating_Runtime_Event_Buffer;
    VIO_Execution_Timeline : ST_Heating_Runtime_Execution_Timeline;
  END_VAR
  VAR
    fbEventManager : FB_Heating_Runtime_Event_Manager;
    fbTimelineObserver : FB_Heating_Runtime_Timeline_Observer;
    fbRootCauseCorrelator : FB_Heating_Runtime_RootCause_Correlator;
    fbReconstructionEngine : FB_Heating_Runtime_Event_Reconstruction_Engine;
    fbStabilityModel : FB_Heating_Runtime_Stability_Model;
    fbOTCascadeCorrelator : FB_Heating_Runtime_OT_Cascade_Correlator;
    fbOTInstabilityPredictor : FB_Heating_Runtime_OT_Instability_Predictor;
    fbPredictiveCorrelation : FB_Heating_Runtime_Predictive_Correlation_Weighting_Engine;
    L_Frame : ST_Heating_Runtime_Execution_Frame;
    L_Runtime_Risk : UINT;
    L_Cascade_Risk : UINT;
    L_Circuit_i : INT;
    L_Circuit_Event_Active : BOOL;
    L_Circuit_Event_Code : UINT;
    L_Circuit_Event_Text : STRING(128);
    L_Phase_Event : ST_Heating_Runtime_Phase_Event;
    L_Anomaly : ST_Heating_Runtime_Anomaly;
    L_Source_Instability_Max : REAL;
    L_Source_Instability_UINT : UINT;
    L_Source_Attention : BOOL;
    L_Source_Oscillation_Trend : BOOL;
    L_Source_Degraded_Trend : BOOL;
    L_Source_Loss_Trend : BOOL;
  END_VAR

            // ==============================================================================
// Heating runtime supervisory enrichment
// Passive observability-only connector for restored supervisory FB stack.
//
// DOES NOT own runtime.
// DOES NOT own heating logic.
// DOES NOT own diagnostics authority.
// DOES NOT own OpenTherm transport.
// DOES NOT write outputs or commands.
// ==============================================================================



// ======================================================
// DEFAULTS
// ======================================================
VO_Status_Code := 0;
VO_Status_Text := 'Heating runtime supervisory enrichment disabled';

IF NOT VI_Enable THEN
    RETURN;
END_IF;

// ======================================================
// PASSIVE CIRCUIT EDGE INGESTION
// ======================================================
// Circuit control publishes canonical runtime projection only. This supervisory
// connector is the integration boundary that raises those passive projection
// edges into the event/anomaly stream used by timeline, reconstruction and
// causality observers.
L_Phase_Event := VI_Phase_Event;
L_Anomaly := VI_Anomaly;
L_Circuit_Event_Active := FALSE;
L_Circuit_Event_Code := 0;
L_Circuit_Event_Text := '';

FOR L_Circuit_i := 1 TO GVL_CONSTANTS.C_MAX_HEATING_CIRCUITS DO
    IF GVL_Heating_Runtime_Projection.G_Circuit_Projection[L_Circuit_i].Source_Loss_Event THEN
        L_Circuit_Event_Active := TRUE;
        L_Circuit_Event_Code := 804;
        L_Circuit_Event_Text := 'Heating circuit temperature source loss';
        EXIT;
    ELSIF GVL_Heating_Runtime_Projection.G_Circuit_Projection[L_Circuit_i].Fallback_Activated_Event THEN
        L_Circuit_Event_Active := TRUE;
        L_Circuit_Event_Code := 802;
        L_Circuit_Event_Text := 'Heating circuit fallback activated';
        EXIT;
    ELSIF GVL_Heating_Runtime_Projection.G_Circuit_Projection[L_Circuit_i].Fallback_Recovered_Event THEN
        L_Circuit_Event_Active := TRUE;
        L_Circuit_Event_Code := 803;
        L_Circuit_Event_Text := 'Heating circuit fallback recovered';
        EXIT;
    ELSIF GVL_Heating_Runtime_Projection.G_Circuit_Projection[L_Circuit_i].Source_Switched_Event THEN
        L_Circuit_Event_Active := TRUE;
        L_Circuit_Event_Code := 801;
        L_Circuit_Event_Text := 'Heating circuit temperature source switched';
        EXIT;
    END_IF;
END_FOR;

IF L_Circuit_Event_Active THEN
    L_Phase_Event.Phase := VI_Runtime_Context.Current_Phase;
    L_Phase_Event.Event_Active := TRUE;
    L_Phase_Event.Event_Completed := TRUE;
    L_Phase_Event.Event_Failed := FALSE;
    L_Phase_Event.Start_Time_MS := VI_System_Time_MS;
    L_Phase_Event.End_Time_MS := VI_System_Time_MS;
    L_Phase_Event.Duration_MS := 0;
    L_Phase_Event.Ordering_Valid := TRUE;
    L_Phase_Event.Isolation_Valid := TRUE;
    L_Phase_Event.Status_Code := L_Circuit_Event_Code;
    L_Phase_Event.Status_Text := L_Circuit_Event_Text;
    L_Phase_Event.Diagnostics_Visible := TRUE;
    L_Phase_Event.Explainability_Visible := TRUE;
    L_Phase_Event.Safety_Integrity_Valid := TRUE;
    L_Phase_Event.OpenTherm_Ownership_Valid := TRUE;
    L_Phase_Event.Cascade_Ownership_Valid := TRUE;

    L_Anomaly.Anomaly_Active := TRUE;
    L_Anomaly.Runtime_Degraded := L_Anomaly.Runtime_Degraded OR (L_Circuit_Event_Code = 802) OR (L_Circuit_Event_Code = 804);
    L_Anomaly.Diagnostics_Degraded := L_Anomaly.Diagnostics_Degraded OR (L_Circuit_Event_Code = 804);
    L_Anomaly.Explainability_Degraded := L_Anomaly.Explainability_Degraded OR (L_Circuit_Event_Code = 804);

    IF L_Circuit_Event_Code = 804 THEN
        IF L_Anomaly.Severity_Level < 80 THEN
            L_Anomaly.Severity_Level := 80;
        END_IF;
        L_Anomaly.Status_Code := 804;
        L_Anomaly.Status_Text := 'Heating circuit source loss observed';
    ELSIF L_Circuit_Event_Code = 802 THEN
        IF L_Anomaly.Severity_Level < 40 THEN
            L_Anomaly.Severity_Level := 40;
        END_IF;
        L_Anomaly.Status_Code := 802;
        L_Anomaly.Status_Text := 'Heating circuit fallback activation observed';
    ELSIF L_Circuit_Event_Code = 803 THEN
        L_Anomaly.Status_Code := 803;
        L_Anomaly.Status_Text := 'Heating circuit fallback recovery observed';
    ELSE
        L_Anomaly.Status_Code := 801;
        L_Anomaly.Status_Text := 'Heating circuit source switch observed';
    END_IF;
END_IF;

// ======================================================
// SOURCE INSTABILITY AGGREGATION
// ======================================================
// Per-circuit predictive details remain in GVL_Heating_Source_Stability.G_State.
// This supervisory layer publishes only the aggregate source-instability view
// into the canonical runtime predictive state.
L_Source_Instability_Max := REAL#0.0;
L_Source_Attention := FALSE;
L_Source_Oscillation_Trend := FALSE;
L_Source_Degraded_Trend := FALSE;
L_Source_Loss_Trend := FALSE;

FOR L_Circuit_i := 1 TO GVL_CONSTANTS.C_MAX_HEATING_CIRCUITS DO
    IF GVL_Heating_Source_Stability.G_State[L_Circuit_i].Instability_Score > L_Source_Instability_Max THEN
        L_Source_Instability_Max := GVL_Heating_Source_Stability.G_State[L_Circuit_i].Instability_Score;
    END_IF;

    L_Source_Attention :=
        L_Source_Attention OR
        GVL_Heating_Source_Stability.G_State[L_Circuit_i].Instability_Attention;

    L_Source_Oscillation_Trend :=
        L_Source_Oscillation_Trend OR
        GVL_Heating_Source_Stability.G_State[L_Circuit_i].Oscillation_Detected;

    L_Source_Degraded_Trend :=
        L_Source_Degraded_Trend OR
        GVL_Heating_Source_Stability.G_State[L_Circuit_i].Degraded_Trend_Visible;

    L_Source_Loss_Trend :=
        L_Source_Loss_Trend OR
        (GVL_Heating_Source_Stability.G_State[L_Circuit_i].Source_Loss_Count > 0);
END_FOR;

IF L_Source_Instability_Max < REAL#0.0 THEN
    L_Source_Instability_UINT := 0;
ELSIF L_Source_Instability_Max > REAL#100.0 THEN
    L_Source_Instability_UINT := 100;
ELSE
    L_Source_Instability_UINT := REAL_TO_UINT(L_Source_Instability_Max);
END_IF;

// ======================================================
// EXECUTION FRAME FROM CURRENT RUNTIME CONTEXT
// ======================================================
L_Frame.Phase := VI_Runtime_Context.Current_Phase;
L_Frame.Frame_Started := TRUE;
L_Frame.Frame_Completed := VI_Runtime_Context.Output_Projection_Executed;
L_Frame.Frame_Failed := VI_Runtime_Context.Runtime_Fault;
L_Frame.Frame_Start_MS := VI_System_Time_MS;
L_Frame.Frame_End_MS := VI_System_Time_MS;
L_Frame.Frame_Duration_MS := 0;

L_Frame.Sequencing_Valid :=
    VI_Runtime_Context.DHW_Before_Heating_Valid AND
    VI_Runtime_Context.State_Publication_Before_Diagnostics_Valid AND
    VI_Runtime_Context.Output_Projection_Last_Valid;

L_Frame.Ownership_Valid :=
    VI_Runtime_Context.OpenTherm_Ownership_Valid AND
    VI_Runtime_Context.Cascade_Ownership_Valid AND
    VI_Runtime_Context.Safety_Isolation_Valid;

L_Frame.Synchronization_Valid :=
    VI_Runtime_Context.Diagnostics_Isolation_Valid AND
    VI_Runtime_Context.Explainability_Isolation_Valid;

L_Frame.Runtime_Jitter_Detected := L_Anomaly.Runtime_Jitter_Detected;
L_Frame.Runtime_Latency_Detected := L_Anomaly.Runtime_Latency_Detected;
L_Frame.Runtime_Degraded := L_Anomaly.Runtime_Degraded;
L_Frame.Status_Code := VI_Runtime_Context.Runtime_Status_Code;
L_Frame.Status_Text := VI_Runtime_Context.Runtime_Status_Text;

fbTimelineObserver(
    VI_Enable := TRUE,
    VI_Frame := L_Frame,
    VIO_Timeline := VIO_Execution_Timeline
);

// ======================================================
// EVENT BUFFER
// ======================================================
fbEventManager(
    VI_Enable := TRUE,
    VI_Event := L_Phase_Event,
    VIO_Buffer := VIO_Event_Buffer
);

// ======================================================
// ROOT-CAUSE / CAUSALITY NODE
// ======================================================
fbRootCauseCorrelator(
    VI_Enable := TRUE,
    VI_Anomaly := L_Anomaly
);

VO_Causality_Node := fbRootCauseCorrelator.VO_Node;

// ======================================================
// CAUSALITY EDGE BUILT FROM NODE STATE
// ======================================================
VO_Causality_Edge.Source_Node_ID := 1;
VO_Causality_Edge.Target_Node_ID := 2;
VO_Causality_Edge.Edge_Active := VO_Causality_Node.Node_Active;
VO_Causality_Edge.Propagation_Detected :=
    VO_Causality_Node.Runtime_Degraded OR
    VO_Causality_Node.Runtime_Fault OR
    VO_Causality_Node.Cascade_Degraded OR
    VO_Causality_Node.OpenTherm_Degraded OR
    VO_Causality_Node.Sequencing_Invalid OR
    VO_Causality_Node.Ownership_Invalid OR
    VO_Causality_Node.Synchronization_Invalid;

VO_Causality_Edge.Runtime_Propagation :=
    VO_Causality_Node.Runtime_Degraded OR VO_Causality_Node.Runtime_Fault;
VO_Causality_Edge.Cascade_Propagation := VO_Causality_Node.Cascade_Degraded;
VO_Causality_Edge.OpenTherm_Propagation := VO_Causality_Node.OpenTherm_Degraded;
VO_Causality_Edge.Diagnostics_Propagation := VO_Causality_Node.Diagnostics_Degraded;
VO_Causality_Edge.Sequencing_Propagation := VO_Causality_Node.Sequencing_Invalid;
VO_Causality_Edge.Ownership_Propagation := VO_Causality_Node.Ownership_Invalid;
VO_Causality_Edge.Synchronization_Propagation := VO_Causality_Node.Synchronization_Invalid;
VO_Causality_Edge.Severity_Level := VO_Causality_Node.Severity_Level;
VO_Causality_Edge.Critical_Path := VO_Causality_Node.Root_Cause_Candidate;
VO_Causality_Edge.Status_Code := VO_Causality_Node.Status_Code;
VO_Causality_Edge.Status_Text := VO_Causality_Node.Status_Text;

// ======================================================
// FORENSIC RECONSTRUCTION
// ======================================================
fbReconstructionEngine(
    VI_Enable := TRUE,
    VI_Node := VO_Causality_Node,
    VI_Edge := VO_Causality_Edge,
    VI_System_Time_MS := VI_System_Time_MS
);

VO_Blackbox_Event := fbReconstructionEngine.VO_Event;

// ======================================================
// STABILITY / OT / CASCADE PREDICTIVE SUPERVISION
// ======================================================
fbStabilityModel(
    VI_Enable := TRUE,
    VI_Runtime_Degraded := L_Anomaly.Runtime_Degraded,
    VI_Runtime_Critical := L_Anomaly.Critical_Anomaly
);

fbOTCascadeCorrelator(
    VI_Enable := TRUE,
    VI_Cascade_Degraded := L_Anomaly.Cascade_Degraded,
    VI_OT_Degraded := L_Anomaly.OpenTherm_Transport_Degraded,
    VI_OT_Command_Valid := VI_OT_Command_Valid,
    VI_Boiler_Count := VI_Cascade_Boiler_Count
);

fbOTInstabilityPredictor(
    VI_Enable := TRUE,
    VI_OT_Degraded := L_Anomaly.OpenTherm_Transport_Degraded,
    VI_OT_Command_Valid := VI_OT_Command_Valid
);

IF L_Anomaly.Critical_Anomaly THEN
    L_Runtime_Risk := 100;
ELSIF L_Anomaly.Runtime_Degraded THEN
    L_Runtime_Risk := 60;
ELSE
    L_Runtime_Risk := 0;
END_IF;

IF L_Anomaly.Cascade_Boiler_Loss_Detected THEN
    L_Cascade_Risk := 100;
ELSIF L_Anomaly.Cascade_Degraded THEN
    L_Cascade_Risk := 60;
ELSE
    L_Cascade_Risk := 0;
END_IF;

fbPredictiveCorrelation(
    VI_Enable := TRUE,
    VI_Runtime_Risk := L_Runtime_Risk,
    VI_Cascade_Risk := L_Cascade_Risk,
    VI_OT_Risk := fbOTInstabilityPredictor.VO_OT_Instability_Risk
);

// ======================================================
// PREDICTIVE PUBLICATION MODEL
// ======================================================
VO_Predictive_State.Predictive_Analytics_Visible := TRUE;
VO_Predictive_State.Predictive_Analytics_Degraded :=
    fbPredictiveCorrelation.VO_Correlation_Degraded OR L_Source_Attention;
VO_Predictive_State.Predictive_Analytics_Attention :=
    (fbPredictiveCorrelation.VO_Correlation_Score > 40) OR L_Source_Attention;
VO_Predictive_State.Runtime_Stable := fbStabilityModel.VO_Runtime_Stable;
VO_Predictive_State.Runtime_Stability_Score := fbStabilityModel.VO_Stability_Score;
VO_Predictive_State.Runtime_Degradation_Observation := L_Runtime_Risk;
VO_Predictive_State.Runtime_Failure_Observation := SEL(L_Anomaly.Critical_Anomaly, 0, 100);
VO_Predictive_State.Source_Instability_Observation := L_Source_Instability_UINT;
VO_Predictive_State.Source_Instability_Attention := L_Source_Attention;
VO_Predictive_State.Source_Oscillation_Trend_Visible := L_Source_Oscillation_Trend;
VO_Predictive_State.Source_Degraded_Trend_Visible := L_Source_Degraded_Trend;
VO_Predictive_State.Source_Loss_Trend_Visible := L_Source_Loss_Trend;
VO_Predictive_State.Cascade_Degradation_Observation := L_Cascade_Risk;
VO_Predictive_State.Cascade_Degraded_Trend_Visible := fbOTCascadeCorrelator.VO_Correlation_Detected;
VO_Predictive_State.OpenTherm_Instability_Observation := fbOTInstabilityPredictor.VO_OT_Instability_Risk;
VO_Predictive_State.OpenTherm_Degraded_Trend_Visible := fbOTInstabilityPredictor.VO_OT_Degraded_Trend;
VO_Predictive_State.Sequencing_Observation := SEL(VO_Causality_Node.Sequencing_Invalid, 0, 100);
VO_Predictive_State.Ownership_Observation := SEL(VO_Causality_Node.Ownership_Invalid, 0, 100);
VO_Predictive_State.Synchronization_Observation := SEL(VO_Causality_Node.Synchronization_Invalid, 0, 100);
VO_Predictive_State.Status_Code := fbPredictiveCorrelation.VO_Status_Code;

IF L_Source_Attention THEN
    VO_Predictive_State.Status_Text := 'Predictive analytics attention: heating source instability observed';
ELSE
    VO_Predictive_State.Status_Text := fbPredictiveCorrelation.VO_Status_Text;
END_IF;

VO_Status_Code := VO_Predictive_State.Status_Code;
VO_Status_Text := VO_Predictive_State.Status_Text;

// >>> BULK_SYNC_ANCHOR: FB_Heating_Runtime_Supervisory_Enrichment <<<
          
END_FUNCTION_BLOCK

FUNCTION_BLOCK FB_Heating_Runtime_OT_Instability_Predictor
  VAR_INPUT
    VI_Enable : BOOL;
    VI_OT_Degraded : BOOL;
    VI_OT_Command_Valid : BOOL;
  END_VAR
  VAR_OUTPUT
    VO_OT_Instability_Risk : UINT;
    VO_OT_Degraded_Trend : BOOL;
    VO_Status_Code : UINT;
    VO_Status_Text : STRING(128);
  END_VAR

            // ==============================================================================
// Heating runtime OT instability predictor
// Read-only predictive OT supervision layer.
// ==============================================================================



VO_OT_Instability_Risk := 0;
VO_OT_Degraded_Trend := FALSE;

VO_Status_Code := 0;
VO_Status_Text := 'Heating runtime OT predictor disabled';

IF NOT VI_Enable THEN
    RETURN;
END_IF;

IF NOT VI_OT_Command_Valid THEN
    VO_OT_Instability_Risk := 100;
    VO_OT_Degraded_Trend := TRUE;

    VO_Status_Code := 900;
    VO_Status_Text := 'Heating runtime OT instability critical';

ELSIF VI_OT_Degraded THEN
    VO_OT_Instability_Risk := 60;
    VO_OT_Degraded_Trend := TRUE;

    VO_Status_Code := 200;
    VO_Status_Text := 'Heating runtime OT degradation trend';

ELSE
    VO_OT_Instability_Risk := 5;

    VO_Status_Code := 1;
    VO_Status_Text := 'Heating runtime OT nominal';
END_IF;

// >>> BULK_SYNC_ANCHOR: FB_Heating_Runtime_OT_Instability_Predictor <<<
          
END_FUNCTION_BLOCK

FUNCTION_BLOCK FB_Presence_Playback
  VAR_INPUT
    VI_Mode_Record : BOOL;
    VI_Time_Index : UDINT;
  END_VAR
  VAR_OUTPUT
    VO_Light_Outputs : ARRAY[1..32] OF BOOL;
  END_VAR
  VAR_IN_OUT
    VI_Light_Inputs : ARRAY[1..32] OF BOOL;
  END_VAR
  VAR
    L_Current_Slot : UDINT;
    L_i : INT;
  END_VAR

            L_Current_Slot := (VI_Time_Index / (GVL_CONSTANTS.C_MS_IN_MINUTE * 10)) MOD TO_UDINT(GVL_CONSTANTS.C_MAX_PRESENCE_HISTORY);

IF VI_Mode_Record THEN
    GVL_Retain.G_Presence_History[L_Current_Slot] := 0;
    FOR L_i := 1 TO 32 DO
        IF VI_Light_Inputs[L_i] THEN
            GVL_Retain.G_Presence_History[L_Current_Slot] := GVL_Retain.G_Presence_History[L_Current_Slot] OR SHL(WORD#1, L_i-1);
        END_IF;
    END_FOR;
ELSE
    FOR L_i := 1 TO 32 DO
        VO_Light_Outputs[L_i] := (GVL_Retain.G_Presence_History[L_Current_Slot] AND SHL(WORD#1, L_i-1)) <> 0;
    END_FOR;
END_IF;
          
END_FUNCTION_BLOCK

FUNCTION_BLOCK FB_Forensic_Journal_Runtime
  VAR_INPUT
    VI_Enable : BOOL;
    VI_System_Time_MS : UDINT;
  END_VAR
  VAR
    L_Record : ST_Forensic_Journal_Record;
    L_Write_Index : UINT;
  END_VAR

            IF NOT VI_Enable THEN
    GVL_Forensic_Journal.G_Runtime_Valid := FALSE;
    RETURN;
END_IF;

L_Write_Index := GVL_Forensic_Journal.G_Write_Index + 1;

IF L_Write_Index > 256 THEN
    L_Write_Index := 1;
END_IF;

IF GVL_Config_Activation.G_Activation_State.Activation_Allowed
   OR GVL_Config_Activation.G_Activation_State.Rollback_Active THEN

    L_Record.Record_Valid := TRUE;
    L_Record.Event_Time_MS := VI_System_Time_MS;
    L_Record.Event_Id := GVL_Forensic_Journal.G_Last_Event_Id + 1;

    L_Record.Config_Version := GVL_Config_Activation.G_Activation_State.Active_Version;
    L_Record.Topology_Version := GVL_Water_Topology_Config.G_Active_Config_Version;

    IF GVL_Config_Activation.G_Activation_State.Rollback_Active THEN
        L_Record.Rollback_Event := TRUE;
        L_Record.Event_Class := 2;
        L_Record.Event_Severity := 2;
        L_Record.Event_Text := 'Topology rollback activated';
        GVL_Forensic_Journal.G_Last_Rollback_Event_Id := L_Record.Event_Id;
    ELSE
        L_Record.Activation_Event := TRUE;
        L_Record.Event_Class := 1;
        L_Record.Event_Severity := 1;
        L_Record.Event_Text := 'Topology activation completed';
        GVL_Forensic_Journal.G_Last_Activation_Event_Id := L_Record.Event_Id;
    END_IF;

    GVL_Forensic_Journal.G_Journal[L_Write_Index] := L_Record;
    GVL_Forensic_Journal.G_Last_Event_Id := L_Record.Event_Id;
    GVL_Forensic_Journal.G_Write_Index := L_Write_Index;
END_IF;

IF GVL_Runtime_Restart_Continuity.G_Continuity_State.Restore_Completed THEN
    L_Write_Index := GVL_Forensic_Journal.G_Write_Index + 1;

    IF L_Write_Index > 256 THEN
        L_Write_Index := 1;
    END_IF;

    L_Record.Record_Valid := TRUE;
    L_Record.Event_Time_MS := VI_System_Time_MS;
    L_Record.Event_Id := GVL_Forensic_Journal.G_Last_Event_Id + 1;
    L_Record.Restart_Event := TRUE;
    L_Record.Event_Class := 3;
    L_Record.Event_Severity := 1;
    L_Record.Config_Version := GVL_Runtime_Restart_Continuity.G_Continuity_State.Active_Config_Version;
    L_Record.Event_Text := 'Warm restart continuity restored';

    GVL_Forensic_Journal.G_Journal[L_Write_Index] := L_Record;
    GVL_Forensic_Journal.G_Last_Event_Id := L_Record.Event_Id;
    GVL_Forensic_Journal.G_Write_Index := L_Write_Index;
    GVL_Forensic_Journal.G_Last_Restart_Event_Id := L_Record.Event_Id;
END_IF;

IF GVL_Config_Activation.G_Config_Quarantine_Active THEN
    L_Write_Index := GVL_Forensic_Journal.G_Write_Index + 1;

    IF L_Write_Index > 256 THEN
        L_Write_Index := 1;
    END_IF;

    L_Record.Record_Valid := TRUE;
    L_Record.Event_Time_MS := VI_System_Time_MS;
    L_Record.Event_Id := GVL_Forensic_Journal.G_Last_Event_Id + 1;
    L_Record.Quarantine_Event := TRUE;
    L_Record.Event_Class := 4;
    L_Record.Event_Severity := 3;
    L_Record.Config_Version := GVL_Config_Activation.G_Activation_State.Staged_Version;
    L_Record.Event_Text := 'Config quarantine active';

    GVL_Forensic_Journal.G_Journal[L_Write_Index] := L_Record;
    GVL_Forensic_Journal.G_Last_Event_Id := L_Record.Event_Id;
    GVL_Forensic_Journal.G_Write_Index := L_Write_Index;
END_IF;

GVL_Forensic_Journal.G_Runtime_Valid := TRUE;
GVL_Forensic_Journal.G_Last_Update_MS := VI_System_Time_MS;
GVL_Forensic_Journal.G_Status_Code := 0;
GVL_Forensic_Journal.G_Status_Text := 'Persistent forensic journal active';
          
END_FUNCTION_BLOCK

